KUKA KRL program: EPS_2_251825_SA38_A_20260116064124.src

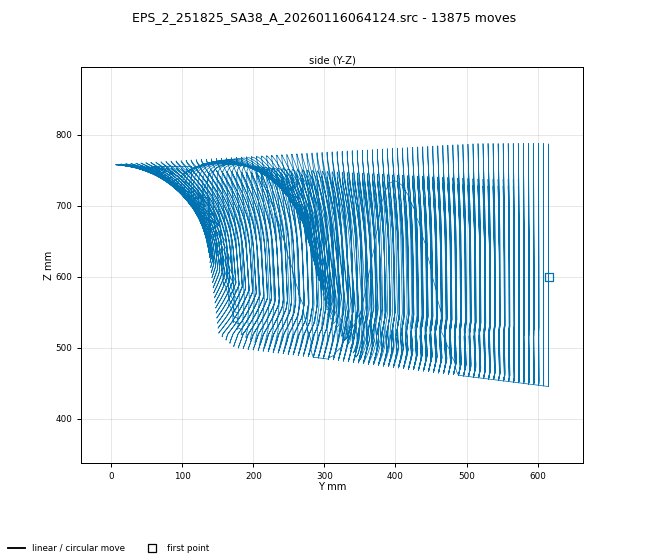
[picture p0: tool path of EPS_2_251825_SA38_A_20260116064124.src, 13875 of 13877 moves have a stored position in this frame; points joined in program order, loops and branches not executed]
&ACCESS RVP
&REL 4
&COMMENT QRS 19112012
&PARAM EDITMASK = *
DEF PART()
EXT BAS (BAS_COMMAND :IN,REAL :IN )
INT I
BAS (#INITMOV,0 )

;KUKA QRS Post kuka4.cps  Date:22-06-2017 !

File_ID=2982

QRS_PRE_INIT()

;Init var - Until changes are made in qrs_pre_init
Outlet_Square_prg=0
Inlet_1_Square_prg=0
Inlet_2_Square_prg=0
Inlet_3_Square_prg=0
Inlet_4_Square_prg=0
Inlet_5_Square_prg=0

Outlet_1={X 0.000, Y 516.340, Z 662.000, B 0.000, E1 0.000 }
Inlet_1={X 0.000, Y 523.470, Z 627.000, B 0.000, E1 180.000 }
Inlet_2={X 0.000, Y 522.780, Z 636.710, B 0.000, E1 270.000 }
Outlet_1_type=251
Inlet_1_type=201
Inlet_2_type=201
;QRS#1=Sidecore dimensions
;QRS#2=250-10" PVC SDR 35
;QRS#3=200-8" PVC SDR 35
;QRS#4=200-8" PVC SDR 35
;QRS#5=
;QRS#6=
;QRS#7=
;QRS#8=
;QRS#9=14M PSX
;QRS#10=12-08 PSX
;QRS#11=12-08 PSX
;QRS#12=
;QRS#13=
;QRS#14=
;QRS#15=
;QRS#16=1220x127x1067 3,5'
;QRS#17=EPS Height
;QRS#18=787,5
;QRS#19=*
;QRS#20= UPDATED VERSION 22-06-2017
;QRS#21=*
Outlet_Square=0100
Inlet_1_Square=0100
Inlet_2_Square=0100
Inlet_3_Square=0
Inlet_4_Square=0
Inlet_5_Square=0
Mill_Square=1
Outlet_Square_Prg=205
Inlet_1_Square_prg=204
Inlet_2_Square_prg=204

QRS_INIT()

$ADVANCE=5

; T1
PTP {E1 173.593,E2 173.593}
PTP {X 0,Y 615.508,A -85,B 0,C 180,E1 173.593,E2 173.593,E3 0,E4 0,E5 0,E6 0}
QRS_SPEED_INIT()
LIN {X 0,Y 615.508,Z 600,A -85,B 0,C 180,E1 173.593,E2 173.593,E3 0,E4 0,E5 0,E6 0} C_VEL
LIN {X 0,Y 615.508,Z 455.497,A -85,B 0,C 180,E1 173.593,E2 173.593} C_VEL
LIN {X 0,Y 615.508,Z 447.326,A -85,B 0,C 180,E1 173.593,E2 173.593} C_VEL
LIN {X 0,Y 615.49,Z 445.326,A -85,B 0,C 180,E1 173.407,E2 173.407} C_VEL
LIN {X 0,Y 615.479,Z 445.312,A -85,B 0,C 180,E1 170.801,E2 170.801} C_VEL
LIN {X 0,Y 615.481,Z 445.31,A -85,B 0,C 180,E1 168.139,E2 168.139} C_VEL
LIN {X 0,Y 615.49,Z 445.327,A -85,B 0,C 180,E1 165.451,E2 165.451} C_VEL
LIN {X 0,Y 615.478,Z 445.31,A -85,B 0,C 180,E1 162.729,E2 162.729} C_VEL
LIN {X 0,Y 615.48,Z 445.314,A -85,B 0,C 180,E1 159.967,E2 159.967} C_VEL
LIN {X 0,Y 615.483,Z 445.318,A -85,B 0,C 180,E1 157.155,E2 157.155} C_VEL
LIN {X 0,Y 615.494,Z 445.306,A -85,B 0,C 180,E1 154.284,E2 154.284} C_VEL
LIN {X 0,Y 615.489,Z 445.322,A -85,B 0,C 180,E1 151.342,E2 151.342} C_VEL
LIN {X 0,Y 615.477,Z 445.313,A -85,B 0,C 180,E1 148.913,E2 148.913} C_VEL
LIN {X 0,Y 615.485,Z 445.307,A -85,B 0,C 180,E1 146.464,E2 146.464} C_VEL
LIN {X 0,Y 615.487,Z 445.325,A -85,B 0,C 180,E1 143.575,E2 143.575} C_VEL
LIN {X 0,Y 615.479,Z 445.313,A -85,B 0,C 180,E1 140.937,E2 140.937} C_VEL
LIN {X 0,Y 615.482,Z 445.308,A -85,B 0,C 180,E1 138.525,E2 138.525} C_VEL
LIN {X 0,Y 615.485,Z 445.317,A -85,B 0,C 180,E1 135.85,E2 135.85} C_VEL
LIN {X 0,Y 615.485,Z 445.313,A -85,B 0,C 180,E1 133.047,E2 133.047} C_VEL
LIN {X 0,Y 615.478,Z 445.309,A -85,B 0,C 180,E1 130.606,E2 130.606} C_VEL
LIN {X 0,Y 615.491,Z 445.312,A -85,B 0,C 180,E1 128.012,E2 128.012} C_VEL
LIN {X 0,Y 615.496,Z 445.324,A -85,B 0,C 180,E1 125.614,E2 125.614} C_VEL
LIN {X 0,Y 615.491,Z 445.316,A -85,B 0,C 180,E1 123.235,E2 123.235} C_VEL
LIN {X 0,Y 615.479,Z 445.312,A -85,B 0,C 180,E1 120.919,E2 120.919} C_VEL
LIN {X 0,Y 615.481,Z 445.309,A -85,B 0,C 180,E1 118.449,E2 118.449} C_VEL
LIN {X 0,Y 615.499,Z 445.325,A -85,B 0,C 180,E1 115.57,E2 115.57} C_VEL
LIN {X 0,Y 615.48,Z 445.31,A -85,B 0,C 180,E1 112.844,E2 112.844} C_VEL
LIN {X 0,Y 615.485,Z 445.416,A -85,B 0,C 180,E1 112.265,E2 112.265} C_VEL
LIN {X 0,Y 615.476,Z 465.419,A -85,B 0,C 180,E1 109.511,E2 109.511} C_VEL
LIN {X 0,Y 615.479,Z 485.735,A -85,B 0,C 180,E1 106.757,E2 106.757} C_VEL
LIN {X 0,Y 615.493,Z 506.841,A -85,B 0,C 180,E1 103.933,E2 103.933} C_VEL
LIN {X 0,Y 615.482,Z 515.432,A -85,B 0,C 180,E1 102.823,E2 102.823} C_VEL
LIN {X 0,Y 615.477,Z 623.203,A -85,B 0,C 180,E1 101.547,E2 101.547} C_VEL
LIN {X 0,Y 615.485,Z 635.76,A -85,B 0,C 180,E1 101.276,E2 101.276} C_VEL
LIN {X 0,Y 615.488,Z 649.105,A -85,B 0,C 180,E1 100.842,E2 100.842} C_VEL
LIN {X 0,Y 615.491,Z 660.086,A -85,B 0,C 180,E1 100.36,E2 100.36} C_VEL
LIN {X 0,Y 615.489,Z 671.819,A -85,B 0,C 180,E1 99.695,E2 99.695} C_VEL
LIN {X 0,Y 615.499,Z 682.28,A -85,B 0,C 180,E1 98.949,E2 98.949} C_VEL
LIN {X 0,Y 615.498,Z 690.84,A -85,B 0,C 180,E1 98.205,E2 98.205} C_VEL
LIN {X 0,Y 615.497,Z 698.718,A -85,B 0,C 180,E1 97.38,E2 97.38} C_VEL
LIN {X 0,Y 615.497,Z 706.405,A -85,B 0,C 180,E1 96.391,E2 96.391} C_VEL
LIN {X 0,Y 615.497,Z 713.463,A -85,B 0,C 180,E1 95.24,E2 95.24} C_VEL
LIN {X 0,Y 615.494,Z 718.162,A -85,B 0,C 180,E1 94.256,E2 94.256} C_VEL
LIN {X 0,Y 615.494,Z 721.757,A -85,B 0,C 180,E1 93.272,E2 93.272} C_VEL
LIN {X 0,Y 615.496,Z 723.617,A -85,B 0,C 180,E1 92.617,E2 92.617} C_VEL
LIN {X 0,Y 615.498,Z 725.035,A -85,B 0,C 180,E1 91.962,E2 91.962} C_VEL
LIN {X 0,Y 615.496,Z 726.642,A -85,B 0,C 180,E1 90.653,E2 90.653} C_VEL
LIN {X 0,Y 615.495,Z 726.884,A -85,B 0,C 180,E1 89.999,E2 89.999} C_VEL
LIN {X 0,Y 615.495,Z 726.705,A -85,B 0,C 180,E1 89.345,E2 89.345} C_VEL
LIN {X 0,Y 615.499,Z 725.181,A -85,B 0,C 180,E1 88.036,E2 88.036} C_VEL
LIN {X 0,Y 615.498,Z 723.839,A -85,B 0,C 180,E1 87.381,E2 87.381} C_VEL
LIN {X 0,Y 615.496,Z 720.991,A -85,B 0,C 180,E1 86.399,E2 86.399} C_VEL
LIN {X 0,Y 615.498,Z 717.131,A -85,B 0,C 180,E1 85.415,E2 85.415} C_VEL
LIN {X 0,Y 615.498,Z 712.147,A -85,B 0,C 180,E1 84.43,E2 84.43} C_VEL
LIN {X 0,Y 615.496,Z 705.708,A -85,B 0,C 180,E1 83.418,E2 83.418} C_VEL
LIN {X 0,Y 615.497,Z 698.03,A -85,B 0,C 180,E1 82.454,E2 82.454} C_VEL
LIN {X 0,Y 615.498,Z 688.25,A -85,B 0,C 180,E1 81.463,E2 81.463} C_VEL
LIN {X 0,Y 615.498,Z 677.982,A -85,B 0,C 180,E1 80.635,E2 80.635} C_VEL
LIN {X 0,Y 615.493,Z 666.416,A -85,B 0,C 180,E1 79.888,E2 79.888} C_VEL
LIN {X 0,Y 615.496,Z 654.517,A -85,B 0,C 180,E1 79.291,E2 79.291} C_VEL
LIN {X 0,Y 615.489,Z 641.636,A -85,B 0,C 180,E1 78.806,E2 78.806} C_VEL
LIN {X 0,Y 615.477,Z 629.028,A -85,B 0,C 180,E1 78.472,E2 78.472} C_VEL
LIN {X 0,Y 615.479,Z 615.873,A -85,B 0,C 180,E1 78.264,E2 78.264} C_VEL
LIN {X 0,Y 615.488,Z 515.092,A -85,B 0,C 180,E1 77.071,E2 77.071} C_VEL
LIN {X 0,Y 615.479,Z 494.007,A -85,B 0,C 180,E1 74.264,E2 74.264} C_VEL
LIN {X 0,Y 615.484,Z 473.933,A -85,B 0,C 180,E1 71.559,E2 71.559} C_VEL
LIN {X 0,Y 615.493,Z 453.348,A -85,B 0,C 180,E1 68.743,E2 68.743} C_VEL
LIN {X 0,Y 615.479,Z 445.31,A -85,B 0,C 180,E1 67.625,E2 67.625} C_VEL
LIN {X 0,Y 615.488,Z 445.309,A -85,B 0,C 180,E1 65.008,E2 65.008} C_VEL
LIN {X 0,Y 615.495,Z 445.317,A -85,B 0,C 180,E1 62.085,E2 62.085} C_VEL
LIN {X 0,Y 615.499,Z 445.31,A -85,B 0,C 180,E1 59.84,E2 59.84} C_VEL
LIN {X 0,Y 615.481,Z 445.309,A -85,B 0,C 180,E1 57.541,E2 57.541} C_VEL
LIN {X 0,Y 615.478,Z 445.309,A -85,B 0,C 180,E1 55.184,E2 55.184} C_VEL
LIN {X 0,Y 615.493,Z 445.312,A -85,B 0,C 180,E1 52.758,E2 52.758} C_VEL
LIN {X 0,Y 615.495,Z 445.313,A -85,B 0,C 180,E1 49.911,E2 49.911} C_VEL
LIN {X 0,Y 615.49,Z 445.308,A -85,B 0,C 180,E1 47.647,E2 47.647} C_VEL
LIN {X 0,Y 615.481,Z 445.311,A -85,B 0,C 180,E1 44.93,E2 44.93} C_VEL
LIN {X 0,Y 615.49,Z 445.319,A -85,B 0,C 180,E1 42.08,E2 42.08} C_VEL
LIN {X 0,Y 615.499,Z 445.308,A -85,B 0,C 180,E1 39.75,E2 39.75} C_VEL
LIN {X 0,Y 615.479,Z 445.312,A -85,B 0,C 180,E1 36.935,E2 36.935} C_VEL
LIN {X 0,Y 615.493,Z 445.313,A -85,B 0,C 180,E1 34.701,E2 34.701} C_VEL
LIN {X 0,Y 615.488,Z 445.31,A -85,B 0,C 180,E1 31.686,E2 31.686} C_VEL
LIN {X 0,Y 615.482,Z 445.308,A -85,B 0,C 180,E1 29.407,E2 29.407} C_VEL
LIN {X 0,Y 615.478,Z 445.31,A -85,B 0,C 180,E1 27.042,E2 27.042} C_VEL
LIN {X 0,Y 615.494,Z 445.325,A -85,B 0,C 180,E1 24.272,E2 24.272} C_VEL
LIN {X 0,Y 615.476,Z 445.317,A -85,B 0,C 180,E1 23.023,E2 23.023} C_VEL
LIN {X 0,Y 615.48,Z 466.086,A -85,B 0,C 180,E1 20.295,E2 20.295} C_VEL
LIN {X 0,Y 615.487,Z 488.175,A -85,B 0,C 180,E1 17.442,E2 17.442} C_VEL
LIN {X 0,Y 615.488,Z 510.904,A -85,B 0,C 180,E1 14.549,E2 14.549} C_VEL
LIN {X 0,Y 615.481,Z 524.429,A -85,B 0,C 180,E1 12.845,E2 12.845} C_VEL
LIN {X 0,Y 615.489,Z 633.994,A -85,B 0,C 180,E1 11.527,E2 11.527} C_VEL
LIN {X 0,Y 615.483,Z 646.945,A -85,B 0,C 180,E1 11.235,E2 11.235} C_VEL
LIN {X 0,Y 615.49,Z 658.842,A -85,B 0,C 180,E1 10.841,E2 10.841} C_VEL
LIN {X 0,Y 615.481,Z 671.405,A -85,B 0,C 180,E1 10.278,E2 10.278} C_VEL
LIN {X 0,Y 615.493,Z 682.784,A -85,B 0,C 180,E1 9.613,E2 9.613} C_VEL
LIN {X 0,Y 615.498,Z 693.031,A -85,B 0,C 180,E1 8.868,E2 8.868} C_VEL
LIN {X 0,Y 615.498,Z 702.243,A -85,B 0,C 180,E1 8.041,E2 8.041} C_VEL
LIN {X 0,Y 615.499,Z 711.101,A -85,B 0,C 180,E1 7.057,E2 7.057} C_VEL
LIN {X 0,Y 615.497,Z 718.333,A -85,B 0,C 180,E1 6.063,E2 6.063} C_VEL
LIN {X 0,Y 615.497,Z 723.167,A -85,B 0,C 180,E1 5.241,E2 5.241} C_VEL
LIN {X 0,Y 615.493,Z 727.867,A -85,B 0,C 180,E1 4.257,E2 4.257} C_VEL
LIN {X 0,Y 615.495,Z 731.464,A -85,B 0,C 180,E1 3.273,E2 3.273} C_VEL
LIN {X 0,Y 615.496,Z 733.324,A -85,B 0,C 180,E1 2.618,E2 2.618} C_VEL
LIN {X 0,Y 615.497,Z 734.743,A -85,B 0,C 180,E1 1.963,E2 1.963} C_VEL
LIN {X 0,Y 615.496,Z 736.351,A -85,B 0,C 180,E1 0.654,E2 0.654} C_VEL
LIN {X 0,Y 615.494,Z 736.594,A -85,B 0,C 180,E1 0,E2 0} C_VEL
LIN {X 0,Y 615.496,Z 736.415,A -85,B 0,C 180,E1 -0.654,E2 -0.654} C_VEL
LIN {X 0,Y 615.496,Z 734.893,A -85,B 0,C 180,E1 -1.963,E2 -1.963} C_VEL
LIN {X 0,Y 615.498,Z 733.551,A -85,B 0,C 180,E1 -2.618,E2 -2.618} C_VEL
LIN {X 0,Y 615.496,Z 730.704,A -85,B 0,C 180,E1 -3.601,E2 -3.601} C_VEL
LIN {X 0,Y 615.499,Z 726.844,A -85,B 0,C 180,E1 -4.584,E2 -4.584} C_VEL
LIN {X 0,Y 615.498,Z 721.862,A -85,B 0,C 180,E1 -5.57,E2 -5.57} C_VEL
LIN {X 0,Y 615.497,Z 715.413,A -85,B 0,C 180,E1 -6.583,E2 -6.583} C_VEL
LIN {X 0,Y 615.497,Z 707.747,A -85,B 0,C 180,E1 -7.545,E2 -7.545} C_VEL
LIN {X 0,Y 615.498,Z 697.969,A -85,B 0,C 180,E1 -8.536,E2 -8.536} C_VEL
LIN {X 0,Y 615.497,Z 687.704,A -85,B 0,C 180,E1 -9.364,E2 -9.364} C_VEL
LIN {X 0,Y 615.476,Z 676.143,A -85,B 0,C 180,E1 -10.111,E2 -10.111} C_VEL
LIN {X 0,Y 615.497,Z 664.291,A -85,B 0,C 180,E1 -10.707,E2 -10.707} C_VEL
LIN {X 0,Y 615.478,Z 651.373,A -85,B 0,C 180,E1 -11.193,E2 -11.193} C_VEL
LIN {X 0,Y 615.486,Z 638.772,A -85,B 0,C 180,E1 -11.527,E2 -11.527} C_VEL
LIN {X 0,Y 615.487,Z 625.651,A -85,B 0,C 180,E1 -11.735,E2 -11.735} C_VEL
LIN {X 0,Y 615.478,Z 524.479,A -85,B 0,C 180,E1 -12.929,E2 -12.929} C_VEL
LIN {X 0,Y 615.488,Z 502.257,A -85,B 0,C 180,E1 -15.735,E2 -15.735} C_VEL
LIN {X 0,Y 615.492,Z 479.506,A -85,B 0,C 180,E1 -18.646,E2 -18.646} C_VEL
LIN {X 0,Y 615.485,Z 456.727,A -85,B 0,C 180,E1 -21.608,E2 -21.608} C_VEL
LIN {X 0,Y 615.476,Z 445.312,A -85,B 0,C 180,E1 -23.134,E2 -23.134} C_VEL
LIN {X 0,Y 615.496,Z 445.309,A -85,B 0,C 180,E1 -25.715,E2 -25.715} C_VEL
LIN {X 0,Y 615.49,Z 445.314,A -85,B 0,C 180,E1 -28.658,E2 -28.658} C_VEL
LIN {X 0,Y 615.477,Z 445.31,A -85,B 0,C 180,E1 -31.084,E2 -31.084} C_VEL
LIN {X 0,Y 615.486,Z 445.312,A -85,B 0,C 180,E1 -33.533,E2 -33.533} C_VEL
LIN {X 0,Y 615.49,Z 445.315,A -85,B 0,C 180,E1 -36.425,E2 -36.425} C_VEL
LIN {X 0,Y 615.479,Z 445.31,A -85,B 0,C 180,E1 -39.06,E2 -39.06} C_VEL
LIN {X 0,Y 615.482,Z 445.315,A -85,B 0,C 180,E1 -41.474,E2 -41.474} C_VEL
LIN {X 0,Y 615.479,Z 445.319,A -85,B 0,C 180,E1 -44.15,E2 -44.15} C_VEL
LIN {X 0,Y 615.486,Z 445.309,A -85,B 0,C 180,E1 -46.953,E2 -46.953} C_VEL
LIN {X 0,Y 615.489,Z 445.32,A -85,B 0,C 180,E1 -49.911,E2 -49.911} C_VEL
LIN {X 0,Y 615.49,Z 445.308,A -85,B 0,C 180,E1 -52.757,E2 -52.757} C_VEL
LIN {X 0,Y 615.488,Z 445.319,A -85,B 0,C 180,E1 -55.299,E2 -55.299} C_VEL
LIN {X 0,Y 615.496,Z 445.32,A -85,B 0,C 180,E1 -57.668,E2 -57.668} C_VEL
LIN {X 0,Y 615.478,Z 445.311,A -85,B 0,C 180,E1 -60.593,E2 -60.593} C_VEL
LIN {X 0,Y 615.496,Z 445.313,A -85,B 0,C 180,E1 -62.954,E2 -62.954} C_VEL
LIN {X 0,Y 615.493,Z 445.313,A -85,B 0,C 180,E1 -65.728,E2 -65.728} C_VEL
LIN {X 0,Y 615.475,Z 445.416,A -85,B 0,C 180,E1 -66.4,E2 -66.4} C_VEL
LIN {X 0,Y 615.49,Z 471.23,A -85,B 0,C 180,E1 -69.094,E2 -69.094} C_VEL
LIN {X 0,Y 615.484,Z 498.445,A -85,B 0,C 180,E1 -71.882,E2 -71.882} C_VEL
LIN {X 0,Y 615.492,Z 523.292,A -85,B 0,C 180,E1 -74.392,E2 -74.392} C_VEL
LIN {X 0,Y 615.484,Z 662.17,A -85,B 0,C 180,E1 -76.05,E2 -76.05} C_VEL
LIN {X 0,Y 615.486,Z 675.829,A -85,B 0,C 180,E1 -76.336,E2 -76.336} C_VEL
LIN {X 0,Y 615.496,Z 689.547,A -85,B 0,C 180,E1 -76.756,E2 -76.756} C_VEL
LIN {X 0,Y 615.497,Z 702.821,A -85,B 0,C 180,E1 -77.302,E2 -77.302} C_VEL
LIN {X 0,Y 615.492,Z 715.587,A -85,B 0,C 180,E1 -77.971,E2 -77.971} C_VEL
LIN {X 0,Y 615.499,Z 727.172,A -85,B 0,C 180,E1 -78.723,E2 -78.723} C_VEL
LIN {X 0,Y 615.498,Z 738.739,A -85,B 0,C 180,E1 -79.639,E2 -79.639} C_VEL
LIN {X 0,Y 615.497,Z 749.081,A -85,B 0,C 180,E1 -80.635,E2 -80.635} C_VEL
LIN {X 0,Y 615.497,Z 757.596,A -85,B 0,C 180,E1 -81.628,E2 -81.628} C_VEL
LIN {X 0,Y 615.496,Z 765.722,A -85,B 0,C 180,E1 -82.784,E2 -82.784} C_VEL
LIN {X 0,Y 615.496,Z 771.426,A -85,B 0,C 180,E1 -83.772,E2 -83.772} C_VEL
LIN {X 0,Y 615.495,Z 776.077,A -85,B 0,C 180,E1 -84.758,E2 -84.758} C_VEL
LIN {X 0,Y 615.494,Z 780.899,A -85,B 0,C 180,E1 -86.071,E2 -86.071} C_VEL
LIN {X 0,Y 615.496,Z 784.25,A -85,B 0,C 180,E1 -87.381,E2 -87.381} C_VEL
LIN {X 0,Y 615.489,Z 786.228,A -85,B 0,C 180,E1 -88.691,E2 -88.691} C_VEL
LIN {X 0,Y 615.493,Z 786.889,A -85,B 0,C 180,E1 -89.999,E2 -89.999} C_VEL
LIN {X 0,Y 615.489,Z 786.23,A -85,B 0,C 180,E1 -91.308,E2 -91.308} C_VEL
LIN {X 0,Y 615.496,Z 784.254,A -85,B 0,C 180,E1 -92.617,E2 -92.617} C_VEL
LIN {X 0,Y 615.493,Z 780.904,A -85,B 0,C 180,E1 -93.928,E2 -93.928} C_VEL
LIN {X 0,Y 615.495,Z 776.084,A -85,B 0,C 180,E1 -95.24,E2 -95.24} C_VEL
LIN {X 0,Y 615.495,Z 769.633,A -85,B 0,C 180,E1 -96.556,E2 -96.556} C_VEL
LIN {X 0,Y 615.497,Z 762.447,A -85,B 0,C 180,E1 -97.709,E2 -97.709} C_VEL
LIN {X 0,Y 615.497,Z 754.911,A -85,B 0,C 180,E1 -98.701,E2 -98.701} C_VEL
LIN {X 0,Y 615.495,Z 745.862,A -85,B 0,C 180,E1 -99.695,E2 -99.695} C_VEL
LIN {X 0,Y 615.497,Z 735.765,A -85,B 0,C 180,E1 -100.617,E2 -100.617} C_VEL
LIN {X 0,Y 615.498,Z 724.871,A -85,B 0,C 180,E1 -101.442,E2 -101.442} C_VEL
LIN {X 0,Y 615.488,Z 712.724,A -85,B 0,C 180,E1 -102.194,E2 -102.194} C_VEL
LIN {X 0,Y 615.495,Z 699.113,A -85,B 0,C 180,E1 -102.864,E2 -102.864} C_VEL
LIN {X 0,Y 615.492,Z 685.864,A -85,B 0,C 180,E1 -103.368,E2 -103.368} C_VEL
LIN {X 0,Y 615.484,Z 672.328,A -85,B 0,C 180,E1 -103.747,E2 -103.747} C_VEL
LIN {X 0,Y 615.486,Z 658.097,A -85,B 0,C 180,E1 -104.008,E2 -104.008} C_VEL
LIN {X 0,Y 615.493,Z 523.098,A -85,B 0,C 180,E1 -105.628,E2 -105.628} C_VEL
LIN {X 0,Y 615.479,Z 495.289,A -85,B 0,C 180,E1 -108.44,E2 -108.44} C_VEL
LIN {X 0,Y 615.496,Z 467.859,A -85,B 0,C 180,E1 -111.255,E2 -111.255} C_VEL
LIN {X 0,Y 615.477,Z 445.31,A -85,B 0,C 180,E1 -113.612,E2 -113.612} C_VEL
LIN {X 0,Y 615.492,Z 445.317,A -85,B 0,C 180,E1 -116.443,E2 -116.443} C_VEL
LIN {X 0,Y 615.493,Z 445.324,A -85,B 0,C 180,E1 -118.656,E2 -118.656} C_VEL
LIN {X 0,Y 615.493,Z 445.314,A -85,B 0,C 180,E1 -121.087,E2 -121.087} C_VEL
LIN {X 0,Y 615.479,Z 445.31,A -85,B 0,C 180,E1 -123.533,E2 -123.533} C_VEL
LIN {X 0,Y 615.477,Z 445.31,A -85,B 0,C 180,E1 -125.832,E2 -125.832} C_VEL
LIN {X 0,Y 615.488,Z 445.31,A -85,B 0,C 180,E1 -128.067,E2 -128.067} C_VEL
LIN {X 0,Y 615.49,Z 445.314,A -85,B 0,C 180,E1 -131.095,E2 -131.095} C_VEL
LIN {X 0,Y 615.499,Z 445.308,A -85,B 0,C 180,E1 -133.242,E2 -133.242} C_VEL
LIN {X 0,Y 615.482,Z 445.31,A -85,B 0,C 180,E1 -136.001,E2 -136.001} C_VEL
LIN {X 0,Y 615.492,Z 445.318,A -85,B 0,C 180,E1 -138.903,E2 -138.903} C_VEL
LIN {X 0,Y 615.487,Z 445.314,A -85,B 0,C 180,E1 -141.096,E2 -141.096} C_VEL
LIN {X 0,Y 615.481,Z 445.308,A -85,B 0,C 180,E1 -143.575,E2 -143.575} C_VEL
LIN {X 0,Y 615.496,Z 445.319,A -85,B 0,C 180,E1 -146.462,E2 -146.462} C_VEL
LIN {X 0,Y 615.49,Z 445.313,A -85,B 0,C 180,E1 -149.08,E2 -149.08} C_VEL
LIN {X 0,Y 615.483,Z 445.308,A -85,B 0,C 180,E1 -151.548,E2 -151.548} C_VEL
LIN {X 0,Y 615.493,Z 445.319,A -85,B 0,C 180,E1 -154.427,E2 -154.427} C_VEL
LIN {X 0,Y 615.486,Z 445.312,A -85,B 0,C 180,E1 -157.155,E2 -157.155} C_VEL
LIN {X 0,Y 615.487,Z 445.308,A -85,B 0,C 180,E1 -159.439,E2 -159.439} C_VEL
LIN {X 0,Y 615.478,Z 445.313,A -85,B 0,C 180,E1 -162.043,E2 -162.043} C_VEL
LIN {X 0,Y 615.489,Z 445.321,A -85,B 0,C 180,E1 -164.774,E2 -164.774} C_VEL
LIN {X 0,Y 615.49,Z 445.307,A -85,B 0,C 180,E1 -167.47,E2 -167.47} C_VEL
LIN {X 0,Y 615.479,Z 445.315,A -85,B 0,C 180,E1 -170.138,E2 -170.138} C_VEL
LIN {X 0,Y 615.486,Z 445.321,A -85,B 0,C 180,E1 -172.784,E2 -172.784} C_VEL
LIN {X 0,Y 615.496,Z 445.306,A -85,B 0,C 180,E1 -175.416,E2 -175.416} C_VEL
LIN {X 0,Y 615.477,Z 445.314,A -85,B 0,C 180,E1 -178.037,E2 -178.037} C_VEL
LIN {X 0,Y 615.488,Z 445.325,A -85,B 0,C 180,E1 -180.654,E2 -180.654} C_VEL
LIN {X 0,Y 615.484,Z 445.31,A -85,B 0,C 180,E1 -183.273,E2 -183.273} C_VEL
LIN {X 0,Y 615.478,Z 445.311,A -85,B 0,C 180,E1 -185.899,E2 -185.899} C_VEL
LIN {X 0,Y 615.49,Z 445.326,A -85,B 0,C 180,E1 -186.593,E2 -186.593} C_VEL
LIN {X 0,Y 614.808,Z 445.46,A -85,B 0,C 180,E1 -187.138,E2 -187.138} C_VEL
LIN {X 0,Y 611.967,Z 445.877,A -85,B 0,C 180,E1 -188.024,E2 -188.024} C_VEL
LIN {X 0,Y 609.574,Z 446.186,A -85,B 0,C 180,E1 -188.737,E2 -188.737} C_VEL
LIN {X 0,Y 608.54,Z 446.303,A -85,B 0,C 180,E1 -189.287,E2 -189.287} C_VEL
LIN {X 0,Y 608.451,Z 446.312,A -85,B 0,C 180,E1 -189.473,E2 -189.473} C_VEL
LIN {X 0,Y 608.458,Z 446.314,A -85,B 0,C 180,E1 -192,E2 -192} C_VEL
LIN {X 0,Y 608.474,Z 446.317,A -85,B 0,C 180,E1 -194.721,E2 -194.721} C_VEL
LIN {X 0,Y 608.445,Z 446.313,A -85,B 0,C 180,E1 -197.477,E2 -197.477} C_VEL
LIN {X 0,Y 608.461,Z 446.317,A -85,B 0,C 180,E1 -200.274,E2 -200.274} C_VEL
LIN {X 0,Y 608.447,Z 446.315,A -85,B 0,C 180,E1 -203.124,E2 -203.124} C_VEL
LIN {X 0,Y 608.476,Z 446.31,A -85,B 0,C 180,E1 -205.725,E2 -205.725} C_VEL
LIN {X 0,Y 608.476,Z 446.318,A -85,B 0,C 180,E1 -208.623,E2 -208.623} C_VEL
LIN {X 0,Y 608.469,Z 446.31,A -85,B 0,C 180,E1 -211.317,E2 -211.317} C_VEL
LIN {X 0,Y 608.471,Z 446.31,A -85,B 0,C 180,E1 -213.737,E2 -213.737} C_VEL
LIN {X 0,Y 608.472,Z 446.314,A -85,B 0,C 180,E1 -216.091,E2 -216.091} C_VEL
LIN {X 0,Y 608.467,Z 446.32,A -85,B 0,C 180,E1 -218.588,E2 -218.588} C_VEL
LIN {X 0,Y 608.456,Z 446.312,A -85,B 0,C 180,E1 -221.344,E2 -221.344} C_VEL
LIN {X 0,Y 608.453,Z 446.319,A -85,B 0,C 180,E1 -224.265,E2 -224.265} C_VEL
LIN {X 0,Y 608.453,Z 446.314,A -85,B 0,C 180,E1 -227.042,E2 -227.042} C_VEL
LIN {X 0,Y 608.453,Z 446.313,A -85,B 0,C 180,E1 -229.698,E2 -229.698} C_VEL
LIN {X 0,Y 608.475,Z 446.317,A -85,B 0,C 180,E1 -232.256,E2 -232.256} C_VEL
LIN {X 0,Y 608.471,Z 446.311,A -85,B 0,C 180,E1 -235.092,E2 -235.092} C_VEL
LIN {X 0,Y 608.47,Z 446.312,A -85,B 0,C 180,E1 -237.907,E2 -237.907} C_VEL
LIN {X 0,Y 608.472,Z 446.317,A -85,B 0,C 180,E1 -240.222,E2 -240.222} C_VEL
LIN {X 0,Y 608.483,Z 446.313,A -85,B 0,C 180,E1 -242.793,E2 -242.793} C_VEL
LIN {X 0,Y 608.455,Z 446.312,A -85,B 0,C 180,E1 -245.43,E2 -245.43} C_VEL
LIN {X 0,Y 608.476,Z 446.356,A -85,B 0,C 180,E1 -247.596,E2 -247.596} C_VEL
LIN {X 0,Y 608.536,Z 462.894,A -85,B 0,C 180,E1 -249.906,E2 -249.906} C_VEL
LIN {X 0,Y 608.527,Z 483.248,A -85,B 0,C 180,E1 -252.7,E2 -252.7} C_VEL
LIN {X 0,Y 608.509,Z 506.148,A -85,B 0,C 180,E1 -255.794,E2 -255.794} C_VEL
LIN {X 0,Y 608.481,Z 515.512,A -85,B 0,C 180,E1 -257.027,E2 -257.027} C_VEL
LIN {X 0,Y 608.541,Z 623.349,A -85,B 0,C 180,E1 -258.32,E2 -258.32} C_VEL
LIN {X 0,Y 608.525,Z 636.65,A -85,B 0,C 180,E1 -258.615,E2 -258.615} C_VEL
LIN {X 0,Y 608.52,Z 649.964,A -85,B 0,C 180,E1 -259.059,E2 -259.059} C_VEL
LIN {X 0,Y 608.501,Z 661.886,A -85,B 0,C 180,E1 -259.604,E2 -259.604} C_VEL
LIN {X 0,Y 608.502,Z 673.304,A -85,B 0,C 180,E1 -260.276,E2 -260.276} C_VEL
LIN {X 0,Y 608.474,Z 683.596,A -85,B 0,C 180,E1 -261.03,E2 -261.03} C_VEL
LIN {X 0,Y 608.464,Z 692.859,A -85,B 0,C 180,E1 -261.867,E2 -261.867} C_VEL
LIN {X 0,Y 608.466,Z 701.831,A -85,B 0,C 180,E1 -262.868,E2 -262.868} C_VEL
LIN {X 0,Y 608.444,Z 709.061,A -85,B 0,C 180,E1 -263.867,E2 -263.867} C_VEL
LIN {X 0,Y 608.462,Z 713.939,A -85,B 0,C 180,E1 -264.699,E2 -264.699} C_VEL
LIN {X 0,Y 608.439,Z 718.682,A -85,B 0,C 180,E1 -265.695,E2 -265.695} C_VEL
LIN {X 0,Y 608.425,Z 722.315,A -85,B 0,C 180,E1 -266.69,E2 -266.69} C_VEL
LIN {X 0,Y 608.425,Z 724.193,A -85,B 0,C 180,E1 -267.353,E2 -267.353} C_VEL
LIN {X 0,Y 608.443,Z 725.628,A -85,B 0,C 180,E1 -268.015,E2 -268.015} C_VEL
LIN {X 0,Y 608.439,Z 727.252,A -85,B 0,C 180,E1 -269.339,E2 -269.339} C_VEL
LIN {X 0,Y 608.435,Z 727.496,A -85,B 0,C 180,E1 -270.001,E2 -270.001} C_VEL
LIN {X 0,Y 608.438,Z 727.314,A -85,B 0,C 180,E1 -270.663,E2 -270.663} C_VEL
LIN {X 0,Y 608.444,Z 725.775,A -85,B 0,C 180,E1 -271.987,E2 -271.987} C_VEL
LIN {X 0,Y 608.426,Z 724.417,A -85,B 0,C 180,E1 -272.649,E2 -272.649} C_VEL
LIN {X 0,Y 608.45,Z 721.539,A -85,B 0,C 180,E1 -273.643,E2 -273.643} C_VEL
LIN {X 0,Y 608.433,Z 717.639,A -85,B 0,C 180,E1 -274.639,E2 -274.639} C_VEL
LIN {X 0,Y 608.449,Z 712.608,A -85,B 0,C 180,E1 -275.635,E2 -275.635} C_VEL
LIN {X 0,Y 608.441,Z 706.289,A -85,B 0,C 180,E1 -276.634,E2 -276.634} C_VEL
LIN {X 0,Y 608.476,Z 698.371,A -85,B 0,C 180,E1 -277.634,E2 -277.634} C_VEL
LIN {X 0,Y 608.472,Z 688.528,A -85,B 0,C 180,E1 -278.637,E2 -278.637} C_VEL
LIN {X 0,Y 608.48,Z 678.203,A -85,B 0,C 180,E1 -279.474,E2 -279.474} C_VEL
LIN {X 0,Y 608.49,Z 666.586,A -85,B 0,C 180,E1 -280.23,E2 -280.23} C_VEL
LIN {X 0,Y 608.528,Z 655.367,A -85,B 0,C 180,E1 -280.803,E2 -280.803} C_VEL
LIN {X 0,Y 608.527,Z 642.838,A -85,B 0,C 180,E1 -281.288,E2 -281.288} C_VEL
LIN {X 0,Y 608.522,Z 630.026,A -85,B 0,C 180,E1 -281.64,E2 -281.64} C_VEL
LIN {X 0,Y 608.533,Z 617.733,A -85,B 0,C 180,E1 -281.851,E2 -281.851} C_VEL
LIN {X 0,Y 608.529,Z 515.793,A -85,B 0,C 180,E1 -283.058,E2 -283.058} C_VEL
LIN {X 0,Y 608.466,Z 515.079,A -85,B 0,C 180,E1 -283.102,E2 -283.102} C_VEL
LIN {X 0,Y 608.488,Z 495.351,A -85,B 0,C 180,E1 -285.75,E2 -285.75} C_VEL
LIN {X 0,Y 608.529,Z 475.149,A -85,B 0,C 180,E1 -288.496,E2 -288.496} C_VEL
LIN {X 0,Y 608.568,Z 454.621,A -85,B 0,C 180,E1 -291.333,E2 -291.333} C_VEL
LIN {X 0,Y 608.465,Z 446.313,A -85,B 0,C 180,E1 -292.527,E2 -292.527} C_VEL
LIN {X 0,Y 608.456,Z 446.312,A -85,B 0,C 180,E1 -294.572,E2 -294.572} C_VEL
LIN {X 0,Y 608.485,Z 446.312,A -85,B 0,C 180,E1 -297.208,E2 -297.208} C_VEL
LIN {X 0,Y 608.477,Z 446.315,A -85,B 0,C 180,E1 -299.973,E2 -299.973} C_VEL
LIN {X 0,Y 608.458,Z 446.312,A -85,B 0,C 180,E1 -302.88,E2 -302.88} C_VEL
LIN {X 0,Y 608.447,Z 446.317,A -85,B 0,C 180,E1 -305.278,E2 -305.278} C_VEL
LIN {X 0,Y 608.477,Z 446.319,A -85,B 0,C 180,E1 -307.746,E2 -307.746} C_VEL
LIN {X 0,Y 608.453,Z 446.313,A -85,B 0,C 180,E1 -310.329,E2 -310.329} C_VEL
LIN {X 0,Y 608.453,Z 446.313,A -85,B 0,C 180,E1 -312.96,E2 -312.96} C_VEL
LIN {X 0,Y 608.462,Z 446.321,A -85,B 0,C 180,E1 -315.736,E2 -315.736} C_VEL
LIN {X 0,Y 608.457,Z 446.311,A -85,B 0,C 180,E1 -318.659,E2 -318.659} C_VEL
LIN {X 0,Y 608.472,Z 446.319,A -85,B 0,C 180,E1 -321.76,E2 -321.76} C_VEL
LIN {X 0,Y 608.449,Z 446.312,A -85,B 0,C 180,E1 -324.723,E2 -324.723} C_VEL
LIN {X 0,Y 608.469,Z 446.317,A -85,B 0,C 180,E1 -327.477,E2 -327.477} C_VEL
LIN {X 0,Y 608.477,Z 446.312,A -85,B 0,C 180,E1 -330.221,E2 -330.221} C_VEL
LIN {X 0,Y 608.473,Z 446.31,A -85,B 0,C 180,E1 -332.795,E2 -332.795} C_VEL
LIN {X 0,Y 608.455,Z 446.318,A -85,B 0,C 180,E1 -335.429,E2 -335.429} C_VEL
LIN {X 0,Y 608.475,Z 446.327,A -85,B 0,C 180,E1 -336.832,E2 -336.832} C_VEL
LIN {X 0,Y 608.584,Z 462.746,A -85,B 0,C 180,E1 -339.023,E2 -339.023} C_VEL
LIN {X 0,Y 608.533,Z 484.192,A -85,B 0,C 180,E1 -341.831,E2 -341.831} C_VEL
LIN {X 0,Y 608.497,Z 505.639,A -85,B 0,C 180,E1 -344.595,E2 -344.595} C_VEL
LIN {X 0,Y 608.488,Z 524.573,A -85,B 0,C 180,E1 -347.005,E2 -347.005} C_VEL
LIN {X 0,Y 608.554,Z 632.98,A -85,B 0,C 180,E1 -348.319,E2 -348.319} C_VEL
LIN {X 0,Y 608.531,Z 646.326,A -85,B 0,C 180,E1 -348.614,E2 -348.614} C_VEL
LIN {X 0,Y 608.511,Z 658.811,A -85,B 0,C 180,E1 -349.026,E2 -349.026} C_VEL
LIN {X 0,Y 608.509,Z 669.944,A -85,B 0,C 180,E1 -349.519,E2 -349.519} C_VEL
LIN {X 0,Y 608.488,Z 681.719,A -85,B 0,C 180,E1 -350.191,E2 -350.191} C_VEL
LIN {X 0,Y 608.485,Z 692.232,A -85,B 0,C 180,E1 -350.946,E2 -350.946} C_VEL
LIN {X 0,Y 608.475,Z 700.843,A -85,B 0,C 180,E1 -351.699,E2 -351.699} C_VEL
LIN {X 0,Y 608.471,Z 708.773,A -85,B 0,C 180,E1 -352.534,E2 -352.534} C_VEL
LIN {X 0,Y 608.468,Z 716.279,A -85,B 0,C 180,E1 -353.497,E2 -353.497} C_VEL
LIN {X 0,Y 608.451,Z 721.819,A -85,B 0,C 180,E1 -354.365,E2 -354.365} C_VEL
LIN {X 0,Y 608.431,Z 726.96,A -85,B 0,C 180,E1 -355.362,E2 -355.362} C_VEL
LIN {X 0,Y 608.45,Z 730.95,A -85,B 0,C 180,E1 -356.358,E2 -356.358} C_VEL
LIN {X 0,Y 608.425,Z 733.901,A -85,B 0,C 180,E1 -357.352,E2 -357.352} C_VEL
LIN {X 0,Y 608.442,Z 735.337,A -85,B 0,C 180,E1 -358.014,E2 -358.014} C_VEL
LIN {X 0,Y 608.439,Z 736.962,A -85,B 0,C 180,E1 -359.338,E2 -359.338} C_VEL
LIN {X 0,Y 608.434,Z 737.205,A -85,B 0,C 180,E1 -360,E2 -360} C_VEL
LIN {X 0,Y 608.439,Z 737.025,A -85,B 0,C 180,E1 -360.662,E2 -360.662} C_VEL
LIN {X 0,Y 608.441,Z 735.486,A -85,B 0,C 180,E1 -361.986,E2 -361.986} C_VEL
LIN {X 0,Y 608.426,Z 734.127,A -85,B 0,C 180,E1 -362.648,E2 -362.648} C_VEL
LIN {X 0,Y 608.449,Z 731.251,A -85,B 0,C 180,E1 -363.642,E2 -363.642} C_VEL
LIN {X 0,Y 608.433,Z 727.351,A -85,B 0,C 180,E1 -364.638,E2 -364.638} C_VEL
LIN {X 0,Y 608.449,Z 722.321,A -85,B 0,C 180,E1 -365.634,E2 -365.634} C_VEL
LIN {X 0,Y 608.442,Z 716.005,A -85,B 0,C 180,E1 -366.633,E2 -366.633} C_VEL
LIN {X 0,Y 608.475,Z 708.089,A -85,B 0,C 180,E1 -367.633,E2 -367.633} C_VEL
LIN {X 0,Y 608.472,Z 698.243,A -85,B 0,C 180,E1 -368.636,E2 -368.636} C_VEL
LIN {X 0,Y 608.48,Z 687.924,A -85,B 0,C 180,E1 -369.473,E2 -369.473} C_VEL
LIN {X 0,Y 608.473,Z 676.312,A -85,B 0,C 180,E1 -370.229,E2 -370.229} C_VEL
LIN {X 0,Y 608.525,Z 665.111,A -85,B 0,C 180,E1 -370.801,E2 -370.801} C_VEL
LIN {X 0,Y 608.527,Z 652.467,A -85,B 0,C 180,E1 -371.29,E2 -371.29} C_VEL
LIN {X 0,Y 608.53,Z 639.767,A -85,B 0,C 180,E1 -371.639,E2 -371.639} C_VEL
LIN {X 0,Y 608.559,Z 627.504,A -85,B 0,C 180,E1 -371.85,E2 -371.85} C_VEL
LIN {X 0,Y 608.466,Z 524.615,A -85,B 0,C 180,E1 -373.08,E2 -373.08} C_VEL
LIN {X 0,Y 608.495,Z 503.661,A -85,B 0,C 180,E1 -375.749,E2 -375.749} C_VEL
LIN {X 0,Y 608.539,Z 482.36,A -85,B 0,C 180,E1 -378.497,E2 -378.497} C_VEL
LIN {X 0,Y 608.561,Z 460.746,A -85,B 0,C 180,E1 -381.332,E2 -381.332} C_VEL
LIN {X 0,Y 608.45,Z 446.328,A -85,B 0,C 180,E1 -383.259,E2 -383.259} C_VEL
LIN {X 0,Y 608.456,Z 446.318,A -85,B 0,C 180,E1 -386.035,E2 -386.035} C_VEL
LIN {X 0,Y 608.479,Z 446.314,A -85,B 0,C 180,E1 -388.62,E2 -388.62} C_VEL
LIN {X 0,Y 608.448,Z 446.313,A -85,B 0,C 180,E1 -391.318,E2 -391.318} C_VEL
LIN {X 0,Y 608.476,Z 446.314,A -85,B 0,C 180,E1 -393.735,E2 -393.735} C_VEL
LIN {X 0,Y 608.482,Z 446.319,A -85,B 0,C 180,E1 -396.09,E2 -396.09} C_VEL
LIN {X 0,Y 608.47,Z 446.312,A -85,B 0,C 180,E1 -398.588,E2 -398.588} C_VEL
LIN {X 0,Y 608.457,Z 446.314,A -85,B 0,C 180,E1 -401.341,E2 -401.341} C_VEL
LIN {X 0,Y 608.45,Z 446.317,A -85,B 0,C 180,E1 -404.263,E2 -404.263} C_VEL
LIN {X 0,Y 608.454,Z 446.313,A -85,B 0,C 180,E1 -407.04,E2 -407.04} C_VEL
LIN {X 0,Y 608.457,Z 446.323,A -85,B 0,C 180,E1 -409.696,E2 -409.696} C_VEL
LIN {X 0,Y 608.471,Z 446.312,A -85,B 0,C 180,E1 -412.253,E2 -412.253} C_VEL
LIN {X 0,Y 608.451,Z 446.316,A -85,B 0,C 180,E1 -415.094,E2 -415.094} C_VEL
LIN {X 0,Y 608.47,Z 446.314,A -85,B 0,C 180,E1 -417.905,E2 -417.905} C_VEL
LIN {X 0,Y 608.461,Z 446.312,A -85,B 0,C 180,E1 -420.219,E2 -420.219} C_VEL
LIN {X 0,Y 608.484,Z 446.311,A -85,B 0,C 180,E1 -422.792,E2 -422.792} C_VEL
LIN {X 0,Y 608.484,Z 446.312,A -85,B 0,C 180,E1 -425.846,E2 -425.846} C_VEL
LIN {X 0,Y 608.499,Z 446.453,A -85,B 0,C 180,E1 -426.224,E2 -426.224} C_VEL
LIN {X 0,Y 608.652,Z 461.065,A -85,B 0,C 180,E1 -427.78,E2 -427.78} C_VEL
LIN {X 0,Y 608.584,Z 486.477,A -85,B 0,C 180,E1 -430.433,E2 -430.433} C_VEL
LIN {X 0,Y 608.546,Z 515.829,A -85,B 0,C 180,E1 -433.447,E2 -433.447} C_VEL
LIN {X 0,Y 608.549,Z 523.326,A -85,B 0,C 180,E1 -434.209,E2 -434.209} C_VEL
LIN {X 0,Y 608.615,Z 662.941,A -85,B 0,C 180,E1 -435.903,E2 -435.903} C_VEL
LIN {X 0,Y 608.583,Z 676.597,A -85,B 0,C 180,E1 -436.199,E2 -436.199} C_VEL
LIN {X 0,Y 608.581,Z 690.69,A -85,B 0,C 180,E1 -436.645,E2 -436.645} C_VEL
LIN {X 0,Y 608.562,Z 702.866,A -85,B 0,C 180,E1 -437.155,E2 -437.155} C_VEL
LIN {X 0,Y 608.516,Z 715.667,A -85,B 0,C 180,E1 -437.831,E2 -437.831} C_VEL
LIN {X 0,Y 608.499,Z 728.459,A -85,B 0,C 180,E1 -438.676,E2 -438.676} C_VEL
LIN {X 0,Y 608.496,Z 738.922,A -85,B 0,C 180,E1 -439.518,E2 -439.518} C_VEL
LIN {X 0,Y 608.479,Z 749.326,A -85,B 0,C 180,E1 -440.526,E2 -440.526} C_VEL
LIN {X 0,Y 608.464,Z 757.907,A -85,B 0,C 180,E1 -441.531,E2 -441.531} C_VEL
LIN {X 0,Y 608.461,Z 766.108,A -85,B 0,C 180,E1 -442.7,E2 -442.7} C_VEL
LIN {X 0,Y 608.443,Z 772.544,A -85,B 0,C 180,E1 -443.83,E2 -443.83} C_VEL
LIN {X 0,Y 608.437,Z 777.959,A -85,B 0,C 180,E1 -445.029,E2 -445.029} C_VEL
LIN {X 0,Y 608.432,Z 781.439,A -85,B 0,C 180,E1 -446.025,E2 -446.025} C_VEL
LIN {X 0,Y 608.424,Z 784.829,A -85,B 0,C 180,E1 -447.351,E2 -447.351} C_VEL
LIN {X 0,Y 608.442,Z 786.829,A -85,B 0,C 180,E1 -448.675,E2 -448.675} C_VEL
LIN {X 0,Y 608.433,Z 787.5,A -85,B 0,C 180,E1 -449.999,E2 -449.999} C_VEL
LIN {X 0,Y 608.442,Z 786.831,A -85,B 0,C 180,E1 -451.323,E2 -451.323} C_VEL
LIN {X 0,Y 608.424,Z 784.833,A -85,B 0,C 180,E1 -452.647,E2 -452.647} C_VEL
LIN {X 0,Y 608.431,Z 781.444,A -85,B 0,C 180,E1 -453.973,E2 -453.973} C_VEL
LIN {X 0,Y 608.44,Z 776.571,A -85,B 0,C 180,E1 -455.301,E2 -455.301} C_VEL
LIN {X 0,Y 608.444,Z 770.216,A -85,B 0,C 180,E1 -456.603,E2 -456.603} C_VEL
LIN {X 0,Y 608.453,Z 762.804,A -85,B 0,C 180,E1 -457.799,E2 -457.799} C_VEL
LIN {X 0,Y 608.472,Z 753.831,A -85,B 0,C 180,E1 -458.97,E2 -458.97} C_VEL
LIN {X 0,Y 608.472,Z 744.401,A -85,B 0,C 180,E1 -459.976,E2 -459.976} C_VEL
LIN {X 0,Y 608.505,Z 733.051,A -85,B 0,C 180,E1 -460.973,E2 -460.973} C_VEL
LIN {X 0,Y 608.532,Z 721.162,A -85,B 0,C 180,E1 -461.828,E2 -461.828} C_VEL
LIN {X 0,Y 608.531,Z 708.09,A -85,B 0,C 180,E1 -462.59,E2 -462.59} C_VEL
LIN {X 0,Y 608.562,Z 695.196,A -85,B 0,C 180,E1 -463.183,E2 -463.183} C_VEL
LIN {X 0,Y 608.585,Z 681.216,A -85,B 0,C 180,E1 -463.672,E2 -463.672} C_VEL
LIN {X 0,Y 608.596,Z 667.505,A -85,B 0,C 180,E1 -464.012,E2 -464.012} C_VEL
LIN {X 0,Y 608.622,Z 651.246,A -85,B 0,C 180,E1 -464.256,E2 -464.256} C_VEL
LIN {X 0,Y 608.549,Z 523.343,A -85,B 0,C 180,E1 -465.789,E2 -465.789} C_VEL
LIN {X 0,Y 608.565,Z 495.714,A -85,B 0,C 180,E1 -468.613,E2 -468.613} C_VEL
LIN {X 0,Y 608.641,Z 469.553,A -85,B 0,C 180,E1 -471.328,E2 -471.328} C_VEL
LIN {X 0,Y 608.671,Z 447.529,A -85,B 0,C 180,E1 -473.655,E2 -473.655} C_VEL
LIN {X 0,Y 608.452,Z 446.314,A -85,B 0,C 180,E1 -473.799,E2 -473.799} C_VEL
LIN {X 0,Y 608.459,Z 446.322,A -85,B 0,C 180,E1 -476.773,E2 -476.773} C_VEL
LIN {X 0,Y 608.47,Z 446.316,A -85,B 0,C 180,E1 -479.018,E2 -479.018} C_VEL
LIN {X 0,Y 608.474,Z 446.311,A -85,B 0,C 180,E1 -481.315,E2 -481.315} C_VEL
LIN {X 0,Y 608.468,Z 446.31,A -85,B 0,C 180,E1 -483.734,E2 -483.734} C_VEL
LIN {X 0,Y 608.473,Z 446.311,A -85,B 0,C 180,E1 -486.089,E2 -486.089} C_VEL
LIN {X 0,Y 608.472,Z 446.319,A -85,B 0,C 180,E1 -488.586,E2 -488.586} C_VEL
LIN {X 0,Y 608.461,Z 446.312,A -85,B 0,C 180,E1 -491.342,E2 -491.342} C_VEL
LIN {X 0,Y 608.46,Z 446.315,A -85,B 0,C 180,E1 -494.264,E2 -494.264} C_VEL
LIN {X 0,Y 608.455,Z 446.316,A -85,B 0,C 180,E1 -497.04,E2 -497.04} C_VEL
LIN {X 0,Y 608.446,Z 446.313,A -85,B 0,C 180,E1 -499.696,E2 -499.696} C_VEL
LIN {X 0,Y 608.466,Z 446.314,A -85,B 0,C 180,E1 -502.253,E2 -502.253} C_VEL
LIN {X 0,Y 608.483,Z 446.312,A -85,B 0,C 180,E1 -505.088,E2 -505.088} C_VEL
LIN {X 0,Y 608.463,Z 446.311,A -85,B 0,C 180,E1 -507.905,E2 -507.905} C_VEL
LIN {X 0,Y 608.472,Z 446.313,A -85,B 0,C 180,E1 -510.221,E2 -510.221} C_VEL
LIN {X 0,Y 608.479,Z 446.317,A -85,B 0,C 180,E1 -512.79,E2 -512.79} C_VEL
LIN {X 0,Y 608.448,Z 446.313,A -85,B 0,C 180,E1 -515.429,E2 -515.429} C_VEL
LIN {X 0,Y 608.471,Z 446.315,A -85,B 0,C 180,E1 -518.309,E2 -518.309} C_VEL
LIN {X 0,Y 608.469,Z 446.311,A -85,B 0,C 180,E1 -521.28,E2 -521.28} C_VEL
LIN {X 0,Y 608.456,Z 446.313,A -85,B 0,C 180,E1 -523.906,E2 -523.906} C_VEL
LIN {X 0,Y 608.463,Z 446.321,A -85,B 0,C 180,E1 -526.644,E2 -526.644} C_VEL
LIN {X 0,Y 608.465,Z 446.311,A -85,B 0,C 180,E1 -529.35,E2 -529.35} C_VEL
LIN {X 0,Y 608.47,Z 446.312,A -85,B 0,C 180,E1 -532.033,E2 -532.033} C_VEL
LIN {X 0,Y 608.466,Z 446.319,A -85,B 0,C 180,E1 -534.698,E2 -534.698} C_VEL
LIN {X 0,Y 608.481,Z 446.309,A -85,B 0,C 180,E1 -537.352,E2 -537.352} C_VEL
LIN {X 0,Y 608.467,Z 446.312,A -85,B 0,C 180,E1 -540,E2 -540} C_VEL
LIN {X 0,Y 608.484,Z 446.318,A -85,B 0,C 180,E1 -542.648,E2 -542.648} C_VEL
LIN {X 0,Y 608.457,Z 446.312,A -85,B 0,C 180,E1 -545.302,E2 -545.302} C_VEL
LIN {X 0,Y 608.471,Z 446.312,A -85,B 0,C 180,E1 -547.967,E2 -547.967} C_VEL
LIN {X 0,Y 608.451,Z 446.312,A -85,B 0,C 180,E1 -549.473,E2 -549.473} C_VEL
LIN {X 0,Y 607.773,Z 446.4,A -85,B 0,C 180,E1 -550.025,E2 -550.025} C_VEL
LIN {X 0,Y 604.92,Z 446.757,A -85,B 0,C 180,E1 -550.922,E2 -550.922} C_VEL
LIN {X 0,Y 602.517,Z 447.056,A -85,B 0,C 180,E1 -551.644,E2 -551.644} C_VEL
LIN {X 0,Y 601.489,Z 447.184,A -85,B 0,C 180,E1 -552.201,E2 -552.201} C_VEL
LIN {X 0,Y 601.406,Z 447.193,A -85,B 0,C 180,E1 -552.389,E2 -552.389} C_VEL
LIN {X 0,Y 601.426,Z 447.192,A -85,B 0,C 180,E1 -554.897,E2 -554.897} C_VEL
LIN {X 0,Y 601.426,Z 447.191,A -85,B 0,C 180,E1 -556.986,E2 -556.986} C_VEL
LIN {X 0,Y 601.402,Z 447.191,A -85,B 0,C 180,E1 -559.81,E2 -559.81} C_VEL
LIN {X 0,Y 601.408,Z 447.199,A -85,B 0,C 180,E1 -562.607,E2 -562.607} C_VEL
LIN {X 0,Y 601.399,Z 447.195,A -85,B 0,C 180,E1 -564.879,E2 -564.879} C_VEL
LIN {X 0,Y 601.419,Z 447.19,A -85,B 0,C 180,E1 -567.868,E2 -567.868} C_VEL
LIN {X 0,Y 601.44,Z 447.19,A -85,B 0,C 180,E1 -570.164,E2 -570.164} C_VEL
LIN {X 0,Y 601.421,Z 447.195,A -85,B 0,C 180,E1 -572.718,E2 -572.718} C_VEL
LIN {X 0,Y 601.415,Z 447.19,A -85,B 0,C 180,E1 -575.117,E2 -575.117} C_VEL
LIN {X 0,Y 601.428,Z 447.187,A -85,B 0,C 180,E1 -577.42,E2 -577.42} C_VEL
LIN {X 0,Y 601.411,Z 447.192,A -85,B 0,C 180,E1 -579.995,E2 -579.995} C_VEL
LIN {X 0,Y 601.407,Z 447.197,A -85,B 0,C 180,E1 -582.671,E2 -582.671} C_VEL
LIN {X 0,Y 601.42,Z 447.188,A -85,B 0,C 180,E1 -585.483,E2 -585.483} C_VEL
LIN {X 0,Y 601.427,Z 447.197,A -85,B 0,C 180,E1 -588.407,E2 -588.407} C_VEL
LIN {X 0,Y 601.434,Z 447.19,A -85,B 0,C 180,E1 -590.877,E2 -590.877} C_VEL
LIN {X 0,Y 601.441,Z 447.186,A -85,B 0,C 180,E1 -593.735,E2 -593.735} C_VEL
LIN {X 0,Y 601.431,Z 447.193,A -85,B 0,C 180,E1 -596.688,E2 -596.688} C_VEL
LIN {X 0,Y 601.431,Z 447.189,A -85,B 0,C 180,E1 -599.06,E2 -599.06} C_VEL
LIN {X 0,Y 601.427,Z 447.188,A -85,B 0,C 180,E1 -601.374,E2 -601.374} C_VEL
LIN {X 0,Y 601.404,Z 447.191,A -85,B 0,C 180,E1 -603.638,E2 -603.638} C_VEL
LIN {X 0,Y 601.423,Z 447.198,A -85,B 0,C 180,E1 -606.591,E2 -606.591} C_VEL
LIN {X 0,Y 601.448,Z 447.307,A -85,B 0,C 180,E1 -607.455,E2 -607.455} C_VEL
LIN {X 0,Y 601.65,Z 456.537,A -85,B 0,C 180,E1 -608.771,E2 -608.771} C_VEL
LIN {X 0,Y 601.569,Z 475.192,A -85,B 0,C 180,E1 -611.378,E2 -611.378} C_VEL
LIN {X 0,Y 601.484,Z 494.702,A -85,B 0,C 180,E1 -614.064,E2 -614.064} C_VEL
LIN {X 0,Y 601.442,Z 513.786,A -85,B 0,C 180,E1 -616.658,E2 -616.658} C_VEL
LIN {X 0,Y 601.486,Z 515.558,A -85,B 0,C 180,E1 -616.874,E2 -616.874} C_VEL
LIN {X 0,Y 601.613,Z 623.379,A -85,B 0,C 180,E1 -618.183,E2 -618.183} C_VEL
LIN {X 0,Y 601.573,Z 636.669,A -85,B 0,C 180,E1 -618.482,E2 -618.482} C_VEL
LIN {X 0,Y 601.537,Z 649.082,A -85,B 0,C 180,E1 -618.896,E2 -618.896} C_VEL
LIN {X 0,Y 601.534,Z 660.268,A -85,B 0,C 180,E1 -619.397,E2 -619.397} C_VEL
LIN {X 0,Y 601.482,Z 672.037,A -85,B 0,C 180,E1 -620.077,E2 -620.077} C_VEL
LIN {X 0,Y 601.444,Z 682.544,A -85,B 0,C 180,E1 -620.84,E2 -620.84} C_VEL
LIN {X 0,Y 601.429,Z 691.15,A -85,B 0,C 180,E1 -621.602,E2 -621.602} C_VEL
LIN {X 0,Y 601.417,Z 699.077,A -85,B 0,C 180,E1 -622.447,E2 -622.447} C_VEL
LIN {X 0,Y 601.376,Z 706.394,A -85,B 0,C 180,E1 -623.394,E2 -623.394} C_VEL
LIN {X 0,Y 601.372,Z 712.118,A -85,B 0,C 180,E1 -624.3,E2 -624.3} C_VEL
LIN {X 0,Y 601.335,Z 717.258,A -85,B 0,C 180,E1 -625.308,E2 -625.308} C_VEL
LIN {X 0,Y 601.367,Z 721.246,A -85,B 0,C 180,E1 -626.316,E2 -626.316} C_VEL
LIN {X 0,Y 601.324,Z 724.195,A -85,B 0,C 180,E1 -627.321,E2 -627.321} C_VEL
LIN {X 0,Y 601.342,Z 725.629,A -85,B 0,C 180,E1 -627.992,E2 -627.992} C_VEL
LIN {X 0,Y 601.339,Z 727.253,A -85,B 0,C 180,E1 -629.331,E2 -629.331} C_VEL
LIN {X 0,Y 601.336,Z 727.496,A -85,B 0,C 180,E1 -630.001,E2 -630.001} C_VEL
LIN {X 0,Y 601.339,Z 727.314,A -85,B 0,C 180,E1 -630.671,E2 -630.671} C_VEL
LIN {X 0,Y 601.343,Z 725.774,A -85,B 0,C 180,E1 -632.01,E2 -632.01} C_VEL
LIN {X 0,Y 601.326,Z 724.415,A -85,B 0,C 180,E1 -632.68,E2 -632.68} C_VEL
LIN {X 0,Y 601.368,Z 721.537,A -85,B 0,C 180,E1 -633.686,E2 -633.686} C_VEL
LIN {X 0,Y 601.337,Z 717.637,A -85,B 0,C 180,E1 -634.694,E2 -634.694} C_VEL
LIN {X 0,Y 601.373,Z 712.605,A -85,B 0,C 180,E1 -635.702,E2 -635.702} C_VEL
LIN {X 0,Y 601.383,Z 706.286,A -85,B 0,C 180,E1 -636.712,E2 -636.712} C_VEL
LIN {X 0,Y 601.397,Z 698.367,A -85,B 0,C 180,E1 -637.724,E2 -637.724} C_VEL
LIN {X 0,Y 601.437,Z 688.521,A -85,B 0,C 180,E1 -638.738,E2 -638.738} C_VEL
LIN {X 0,Y 601.449,Z 678.197,A -85,B 0,C 180,E1 -639.586,E2 -639.586} C_VEL
LIN {X 0,Y 601.492,Z 666.576,A -85,B 0,C 180,E1 -640.35,E2 -640.35} C_VEL
LIN {X 0,Y 601.551,Z 655.356,A -85,B 0,C 180,E1 -640.929,E2 -640.929} C_VEL
LIN {X 0,Y 601.557,Z 642.801,A -85,B 0,C 180,E1 -641.421,E2 -641.421} C_VEL
LIN {X 0,Y 601.587,Z 630.003,A -85,B 0,C 180,E1 -641.776,E2 -641.776} C_VEL
LIN {X 0,Y 601.6,Z 617.694,A -85,B 0,C 180,E1 -641.99,E2 -641.99} C_VEL
LIN {X 0,Y 601.642,Z 516.642,A -85,B 0,C 180,E1 -643.2,E2 -643.2} C_VEL
LIN {X 0,Y 601.468,Z 515.075,A -85,B 0,C 180,E1 -643.257,E2 -643.257} C_VEL
LIN {X 0,Y 601.498,Z 494.074,A -85,B 0,C 180,E1 -646.112,E2 -646.112} C_VEL
LIN {X 0,Y 601.565,Z 475.837,A -85,B 0,C 180,E1 -648.622,E2 -648.622} C_VEL
LIN {X 0,Y 601.664,Z 454.616,A -85,B 0,C 180,E1 -651.59,E2 -651.59} C_VEL
LIN {X 0,Y 601.418,Z 447.202,A -85,B 0,C 180,E1 -652.652,E2 -652.652} C_VEL
LIN {X 0,Y 601.407,Z 447.191,A -85,B 0,C 180,E1 -654.879,E2 -654.879} C_VEL
LIN {X 0,Y 601.425,Z 447.196,A -85,B 0,C 180,E1 -657.868,E2 -657.868} C_VEL
LIN {X 0,Y 601.435,Z 447.19,A -85,B 0,C 180,E1 -660.164,E2 -660.164} C_VEL
LIN {X 0,Y 601.422,Z 447.188,A -85,B 0,C 180,E1 -662.715,E2 -662.715} C_VEL
LIN {X 0,Y 601.398,Z 447.193,A -85,B 0,C 180,E1 -665.112,E2 -665.112} C_VEL
LIN {X 0,Y 601.441,Z 447.192,A -85,B 0,C 180,E1 -667.419,E2 -667.419} C_VEL
LIN {X 0,Y 601.417,Z 447.194,A -85,B 0,C 180,E1 -669.995,E2 -669.995} C_VEL
LIN {X 0,Y 601.416,Z 447.189,A -85,B 0,C 180,E1 -672.671,E2 -672.671} C_VEL
LIN {X 0,Y 601.432,Z 447.194,A -85,B 0,C 180,E1 -675.482,E2 -675.482} C_VEL
LIN {X 0,Y 601.425,Z 447.188,A -85,B 0,C 180,E1 -678.408,E2 -678.408} C_VEL
LIN {X 0,Y 601.415,Z 447.189,A -85,B 0,C 180,E1 -680.873,E2 -680.873} C_VEL
LIN {X 0,Y 601.448,Z 447.195,A -85,B 0,C 180,E1 -683.734,E2 -683.734} C_VEL
LIN {X 0,Y 601.431,Z 447.187,A -85,B 0,C 180,E1 -686.686,E2 -686.686} C_VEL
LIN {X 0,Y 601.417,Z 447.19,A -85,B 0,C 180,E1 -689.058,E2 -689.058} C_VEL
LIN {X 0,Y 601.439,Z 447.191,A -85,B 0,C 180,E1 -691.373,E2 -691.373} C_VEL
LIN {X 0,Y 601.421,Z 447.192,A -85,B 0,C 180,E1 -694.132,E2 -694.132} C_VEL
LIN {X 0,Y 601.468,Z 447.337,A -85,B 0,C 180,E1 -696.683,E2 -696.683} C_VEL
LIN {X 0,Y 601.718,Z 452.894,A -85,B 0,C 180,E1 -697.446,E2 -697.446} C_VEL
LIN {X 0,Y 601.629,Z 474.813,A -85,B 0,C 180,E1 -700.376,E2 -700.376} C_VEL
LIN {X 0,Y 601.55,Z 496.174,A -85,B 0,C 180,E1 -703.181,E2 -703.181} C_VEL
LIN {X 0,Y 601.485,Z 518.097,A -85,B 0,C 180,E1 -706.019,E2 -706.019} C_VEL
LIN {X 0,Y 601.459,Z 524.577,A -85,B 0,C 180,E1 -706.85,E2 -706.85} C_VEL
LIN {X 0,Y 601.674,Z 530.535,A -85,B 0,C 180,E1 -706.941,E2 -706.941} C_VEL
LIN {X 0,Y 601.627,Z 632.969,A -85,B 0,C 180,E1 -708.182,E2 -708.182} C_VEL
LIN {X 0,Y 601.581,Z 646.353,A -85,B 0,C 180,E1 -708.481,E2 -708.481} C_VEL
LIN {X 0,Y 601.552,Z 659.627,A -85,B 0,C 180,E1 -708.928,E2 -708.928} C_VEL
LIN {X 0,Y 601.507,Z 671.576,A -85,B 0,C 180,E1 -709.481,E2 -709.481} C_VEL
LIN {X 0,Y 601.47,Z 683.004,A -85,B 0,C 180,E1 -710.16,E2 -710.16} C_VEL
LIN {X 0,Y 601.438,Z 693.299,A -85,B 0,C 180,E1 -710.923,E2 -710.923} C_VEL
LIN {X 0,Y 601.411,Z 702.562,A -85,B 0,C 180,E1 -711.77,E2 -711.77} C_VEL
LIN {X 0,Y 601.389,Z 711.534,A -85,B 0,C 180,E1 -712.783,E2 -712.783} C_VEL
LIN {X 0,Y 601.376,Z 718.67,A -85,B 0,C 180,E1 -713.781,E2 -713.781} C_VEL
LIN {X 0,Y 601.373,Z 723.64,A -85,B 0,C 180,E1 -714.635,E2 -714.635} C_VEL
LIN {X 0,Y 601.353,Z 728.383,A -85,B 0,C 180,E1 -715.643,E2 -715.643} C_VEL
LIN {X 0,Y 601.345,Z 732.02,A -85,B 0,C 180,E1 -716.65,E2 -716.65} C_VEL
LIN {X 0,Y 601.324,Z 733.903,A -85,B 0,C 180,E1 -717.32,E2 -717.32} C_VEL
LIN {X 0,Y 601.341,Z 735.338,A -85,B 0,C 180,E1 -717.991,E2 -717.991} C_VEL
LIN {X 0,Y 601.339,Z 736.963,A -85,B 0,C 180,E1 -719.33,E2 -719.33} C_VEL
LIN {X 0,Y 601.335,Z 737.206,A -85,B 0,C 180,E1 -720,E2 -720} C_VEL
LIN {X 0,Y 601.339,Z 737.026,A -85,B 0,C 180,E1 -720.67,E2 -720.67} C_VEL
LIN {X 0,Y 601.34,Z 735.487,A -85,B 0,C 180,E1 -722.009,E2 -722.009} C_VEL
LIN {X 0,Y 601.326,Z 734.119,A -85,B 0,C 180,E1 -722.679,E2 -722.679} C_VEL
LIN {X 0,Y 601.368,Z 731.244,A -85,B 0,C 180,E1 -723.685,E2 -723.685} C_VEL
LIN {X 0,Y 601.337,Z 727.343,A -85,B 0,C 180,E1 -724.693,E2 -724.693} C_VEL
LIN {X 0,Y 601.373,Z 722.314,A -85,B 0,C 180,E1 -725.701,E2 -725.701} C_VEL
LIN {X 0,Y 601.383,Z 716.001,A -85,B 0,C 180,E1 -726.711,E2 -726.711} C_VEL
LIN {X 0,Y 601.396,Z 708.086,A -85,B 0,C 180,E1 -727.723,E2 -727.723} C_VEL
LIN {X 0,Y 601.422,Z 700.02,A -85,B 0,C 180,E1 -728.568,E2 -728.568} C_VEL
LIN {X 0,Y 601.453,Z 690.18,A -85,B 0,C 180,E1 -729.415,E2 -729.415} C_VEL
LIN {X 0,Y 601.478,Z 679.129,A -85,B 0,C 180,E1 -730.179,E2 -730.179} C_VEL
LIN {X 0,Y 601.532,Z 666.734,A -85,B 0,C 180,E1 -730.851,E2 -730.851} C_VEL
LIN {X 0,Y 601.553,Z 654.933,A -85,B 0,C 180,E1 -731.339,E2 -731.339} C_VEL
LIN {X 0,Y 601.574,Z 642.479,A -85,B 0,C 180,E1 -731.712,E2 -731.712} C_VEL
LIN {X 0,Y 601.618,Z 628.973,A -85,B 0,C 180,E1 -731.967,E2 -731.967} C_VEL
LIN {X 0,Y 601.561,Z 525.526,A -85,B 0,C 180,E1 -733.212,E2 -733.212} C_VEL
LIN {X 0,Y 601.452,Z 524.611,A -85,B 0,C 180,E1 -733.235,E2 -733.235} C_VEL
LIN {X 0,Y 601.524,Z 503.657,A -85,B 0,C 180,E1 -735.936,E2 -735.936} C_VEL
LIN {X 0,Y 601.582,Z 481.259,A -85,B 0,C 180,E1 -738.864,E2 -738.864} C_VEL
LIN {X 0,Y 601.679,Z 459.4,A -85,B 0,C 180,E1 -741.769,E2 -741.769} C_VEL
LIN {X 0,Y 601.694,Z 448.671,A -85,B 0,C 180,E1 -743.217,E2 -743.217} C_VEL
LIN {X 0,Y 601.429,Z 447.192,A -85,B 0,C 180,E1 -743.456,E2 -743.456} C_VEL
LIN {X 0,Y 601.408,Z 447.2,A -85,B 0,C 180,E1 -746.363,E2 -746.363} C_VEL
LIN {X 0,Y 601.443,Z 447.188,A -85,B 0,C 180,E1 -748.789,E2 -748.789} C_VEL
LIN {X 0,Y 601.424,Z 447.19,A -85,B 0,C 180,E1 -751.454,E2 -751.454} C_VEL
LIN {X 0,Y 601.435,Z 447.197,A -85,B 0,C 180,E1 -754.118,E2 -754.118} C_VEL
LIN {X 0,Y 601.412,Z 447.192,A -85,B 0,C 180,E1 -756.582,E2 -756.582} C_VEL
LIN {X 0,Y 601.416,Z 447.19,A -85,B 0,C 180,E1 -759.126,E2 -759.126} C_VEL
LIN {X 0,Y 601.426,Z 447.196,A -85,B 0,C 180,E1 -761.765,E2 -761.765} C_VEL
LIN {X 0,Y 601.401,Z 447.192,A -85,B 0,C 180,E1 -764.532,E2 -764.532} C_VEL
LIN {X 0,Y 601.455,Z 447.186,A -85,B 0,C 180,E1 -766.425,E2 -766.425} C_VEL
LIN {X 0,Y 601.417,Z 447.195,A -85,B 0,C 180,E1 -769.427,E2 -769.427} C_VEL
LIN {X 0,Y 601.424,Z 447.197,A -85,B 0,C 180,E1 -771.732,E2 -771.732} C_VEL
LIN {X 0,Y 601.388,Z 447.194,A -85,B 0,C 180,E1 -774.245,E2 -774.245} C_VEL
LIN {X 0,Y 601.421,Z 447.189,A -85,B 0,C 180,E1 -776.685,E2 -776.685} C_VEL
LIN {X 0,Y 601.42,Z 447.193,A -85,B 0,C 180,E1 -779.057,E2 -779.057} C_VEL
LIN {X 0,Y 601.438,Z 447.197,A -85,B 0,C 180,E1 -781.373,E2 -781.373} C_VEL
LIN {X 0,Y 601.406,Z 447.197,A -85,B 0,C 180,E1 -783.636,E2 -783.636} C_VEL
LIN {X 0,Y 601.457,Z 447.3,A -85,B 0,C 180,E1 -786.019,E2 -786.019} C_VEL
LIN {X 0,Y 601.863,Z 450.9,A -85,B 0,C 180,E1 -786.425,E2 -786.425} C_VEL
LIN {X 0,Y 601.759,Z 476.202,A -85,B 0,C 180,E1 -789.12,E2 -789.12} C_VEL
LIN {X 0,Y 601.638,Z 501.725,A -85,B 0,C 180,E1 -791.791,E2 -791.791} C_VEL
LIN {X 0,Y 601.568,Z 523.326,A -85,B 0,C 180,E1 -794.021,E2 -794.021} C_VEL
LIN {X 0,Y 601.843,Z 528.553,A -85,B 0,C 180,E1 -794.094,E2 -794.094} C_VEL
LIN {X 0,Y 601.721,Z 662.941,A -85,B 0,C 180,E1 -795.738,E2 -795.738} C_VEL
LIN {X 0,Y 601.693,Z 677.049,A -85,B 0,C 180,E1 -796.05,E2 -796.05} C_VEL
LIN {X 0,Y 601.667,Z 690.691,A -85,B 0,C 180,E1 -796.489,E2 -796.489} C_VEL
LIN {X 0,Y 601.607,Z 704.617,A -85,B 0,C 180,E1 -797.089,E2 -797.089} C_VEL
LIN {X 0,Y 601.546,Z 717.08,A -85,B 0,C 180,E1 -797.774,E2 -797.774} C_VEL
LIN {X 0,Y 601.505,Z 728.461,A -85,B 0,C 180,E1 -798.542,E2 -798.542} C_VEL
LIN {X 0,Y 601.482,Z 738.923,A -85,B 0,C 180,E1 -799.395,E2 -799.395} C_VEL
LIN {X 0,Y 601.43,Z 749.326,A -85,B 0,C 180,E1 -800.414,E2 -800.414} C_VEL
LIN {X 0,Y 601.407,Z 757.907,A -85,B 0,C 180,E1 -801.43,E2 -801.43} C_VEL
LIN {X 0,Y 601.392,Z 766.109,A -85,B 0,C 180,E1 -802.613,E2 -802.613} C_VEL
LIN {X 0,Y 601.361,Z 771.751,A -85,B 0,C 180,E1 -803.604,E2 -803.604} C_VEL
LIN {X 0,Y 601.355,Z 776.564,A -85,B 0,C 180,E1 -804.634,E2 -804.634} C_VEL
LIN {X 0,Y 601.343,Z 781.439,A -85,B 0,C 180,E1 -805.978,E2 -805.978} C_VEL
LIN {X 0,Y 601.323,Z 784.829,A -85,B 0,C 180,E1 -807.32,E2 -807.32} C_VEL
LIN {X 0,Y 601.342,Z 786.83,A -85,B 0,C 180,E1 -808.66,E2 -808.66} C_VEL
LIN {X 0,Y 601.333,Z 787.5,A -85,B 0,C 180,E1 -809.999,E2 -809.999} C_VEL
LIN {X 0,Y 601.342,Z 786.832,A -85,B 0,C 180,E1 -811.338,E2 -811.338} C_VEL
LIN {X 0,Y 601.323,Z 784.833,A -85,B 0,C 180,E1 -812.679,E2 -812.679} C_VEL
LIN {X 0,Y 601.343,Z 781.445,A -85,B 0,C 180,E1 -814.02,E2 -814.02} C_VEL
LIN {X 0,Y 601.354,Z 776.571,A -85,B 0,C 180,E1 -815.364,E2 -815.364} C_VEL
LIN {X 0,Y 601.371,Z 770.626,A -85,B 0,C 180,E1 -816.604,E2 -816.604} C_VEL
LIN {X 0,Y 601.385,Z 763.925,A -85,B 0,C 180,E1 -817.723,E2 -817.723} C_VEL
LIN {X 0,Y 601.411,Z 755.206,A -85,B 0,C 180,E1 -818.906,E2 -818.906} C_VEL
LIN {X 0,Y 601.432,Z 746.091,A -85,B 0,C 180,E1 -819.924,E2 -819.924} C_VEL
LIN {X 0,Y 601.496,Z 735.831,A -85,B 0,C 180,E1 -820.876,E2 -820.876} C_VEL
LIN {X 0,Y 601.533,Z 724.984,A -85,B 0,C 180,E1 -821.711,E2 -821.711} C_VEL
LIN {X 0,Y 601.575,Z 712.794,A -85,B 0,C 180,E1 -822.481,E2 -822.481} C_VEL
LIN {X 0,Y 601.629,Z 701.115,A -85,B 0,C 180,E1 -823.08,E2 -823.08} C_VEL
LIN {X 0,Y 601.651,Z 688.961,A -85,B 0,C 180,E1 -823.577,E2 -823.577} C_VEL
LIN {X 0,Y 601.683,Z 675.045,A -85,B 0,C 180,E1 -824.005,E2 -824.005} C_VEL
LIN {X 0,Y 601.74,Z 660.97,A -85,B 0,C 180,E1 -824.294,E2 -824.294} C_VEL
LIN {X 0,Y 601.728,Z 524.343,A -85,B 0,C 180,E1 -825.961,E2 -825.961} C_VEL
LIN {X 0,Y 601.567,Z 523.343,A -85,B 0,C 180,E1 -825.977,E2 -825.977} C_VEL
LIN {X 0,Y 601.645,Z 496.503,A -85,B 0,C 180,E1 -828.753,E2 -828.753} C_VEL
LIN {X 0,Y 601.777,Z 471.247,A -85,B 0,C 180,E1 -831.404,E2 -831.404} C_VEL
LIN {X 0,Y 601.848,Z 449.223,A -85,B 0,C 180,E1 -833.756,E2 -833.756} C_VEL
LIN {X 0,Y 601.452,Z 447.19,A -85,B 0,C 180,E1 -834.002,E2 -834.002} C_VEL
LIN {X 0,Y 601.456,Z 447.188,A -85,B 0,C 180,E1 -837.11,E2 -837.11} C_VEL
LIN {X 0,Y 601.415,Z 447.19,A -85,B 0,C 180,E1 -839.392,E2 -839.392} C_VEL
LIN {X 0,Y 601.413,Z 447.189,A -85,B 0,C 180,E1 -841.725,E2 -841.725} C_VEL
LIN {X 0,Y 601.428,Z 447.189,A -85,B 0,C 180,E1 -844.117,E2 -844.117} C_VEL
LIN {X 0,Y 601.414,Z 447.197,A -85,B 0,C 180,E1 -846.581,E2 -846.581} C_VEL
LIN {X 0,Y 601.436,Z 447.187,A -85,B 0,C 180,E1 -849.535,E2 -849.535} C_VEL
LIN {X 0,Y 601.436,Z 447.195,A -85,B 0,C 180,E1 -852.593,E2 -852.593} C_VEL
LIN {X 0,Y 601.418,Z 447.189,A -85,B 0,C 180,E1 -855.481,E2 -855.481} C_VEL
LIN {X 0,Y 601.424,Z 447.193,A -85,B 0,C 180,E1 -858.405,E2 -858.405} C_VEL
LIN {X 0,Y 601.435,Z 447.193,A -85,B 0,C 180,E1 -860.875,E2 -860.875} C_VEL
LIN {X 0,Y 601.437,Z 447.185,A -85,B 0,C 180,E1 -863.733,E2 -863.733} C_VEL
LIN {X 0,Y 601.432,Z 447.188,A -85,B 0,C 180,E1 -866.062,E2 -866.062} C_VEL
LIN {X 0,Y 601.436,Z 447.195,A -85,B 0,C 180,E1 -868.54,E2 -868.54} C_VEL
LIN {X 0,Y 601.431,Z 447.187,A -85,B 0,C 180,E1 -871.373,E2 -871.373} C_VEL
LIN {X 0,Y 601.415,Z 447.191,A -85,B 0,C 180,E1 -874.129,E2 -874.129} C_VEL
LIN {X 0,Y 601.419,Z 447.198,A -85,B 0,C 180,E1 -876.59,E2 -876.59} C_VEL
LIN {X 0,Y 601.428,Z 447.187,A -85,B 0,C 180,E1 -879.478,E2 -879.478} C_VEL
LIN {X 0,Y 601.397,Z 447.196,A -85,B 0,C 180,E1 -882.312,E2 -882.312} C_VEL
LIN {X 0,Y 601.428,Z 447.19,A -85,B 0,C 180,E1 -885.103,E2 -885.103} C_VEL
LIN {X 0,Y 601.414,Z 447.19,A -85,B 0,C 180,E1 -887.858,E2 -887.858} C_VEL
LIN {X 0,Y 601.416,Z 447.199,A -85,B 0,C 180,E1 -890.584,E2 -890.584} C_VEL
LIN {X 0,Y 601.444,Z 447.186,A -85,B 0,C 180,E1 -893.323,E2 -893.323} C_VEL
LIN {X 0,Y 601.399,Z 447.192,A -85,B 0,C 180,E1 -895.979,E2 -895.979} C_VEL
LIN {X 0,Y 601.427,Z 447.197,A -85,B 0,C 180,E1 -898.661,E2 -898.661} C_VEL
LIN {X 0,Y 601.422,Z 447.188,A -85,B 0,C 180,E1 -901.339,E2 -901.339} C_VEL
LIN {X 0,Y 601.427,Z 447.187,A -85,B 0,C 180,E1 -903.35,E2 -903.35} C_VEL
LIN {X 0,Y 601.406,Z 447.192,A -85,B 0,C 180,E1 -906.037,E2 -906.037} C_VEL
LIN {X 0,Y 601.435,Z 447.194,A -85,B 0,C 180,E1 -908.738,E2 -908.738} C_VEL
LIN {X 0,Y 601.426,Z 447.187,A -85,B 0,C 180,E1 -911.458,E2 -911.458} C_VEL
LIN {X 0,Y 601.406,Z 447.193,A -85,B 0,C 180,E1 -912.389,E2 -912.389} C_VEL
LIN {X 0,Y 600.743,Z 447.278,A -85,B 0,C 180,E1 -912.948,E2 -912.948} C_VEL
LIN {X 0,Y 597.891,Z 447.632,A -85,B 0,C 180,E1 -913.856,E2 -913.856} C_VEL
LIN {X 0,Y 595.479,Z 447.939,A -85,B 0,C 180,E1 -914.586,E2 -914.586} C_VEL
LIN {X 0,Y 594.441,Z 448.06,A -85,B 0,C 180,E1 -915.15,E2 -915.15} C_VEL
LIN {X 0,Y 594.356,Z 448.069,A -85,B 0,C 180,E1 -915.341,E2 -915.341} C_VEL
LIN {X 0,Y 594.374,Z 448.067,A -85,B 0,C 180,E1 -917.905,E2 -917.905} C_VEL
LIN {X 0,Y 594.377,Z 448.069,A -85,B 0,C 180,E1 -920.92,E2 -920.92} C_VEL
LIN {X 0,Y 594.386,Z 448.065,A -85,B 0,C 180,E1 -923.704,E2 -923.704} C_VEL
LIN {X 0,Y 594.381,Z 448.072,A -85,B 0,C 180,E1 -926.7,E2 -926.7} C_VEL
LIN {X 0,Y 594.38,Z 448.068,A -85,B 0,C 180,E1 -928.999,E2 -928.999} C_VEL
LIN {X 0,Y 594.386,Z 448.065,A -85,B 0,C 180,E1 -931.647,E2 -931.647} C_VEL
LIN {X 0,Y 594.393,Z 448.073,A -85,B 0,C 180,E1 -934.579,E2 -934.579} C_VEL
LIN {X 0,Y 594.379,Z 448.067,A -85,B 0,C 180,E1 -937.087,E2 -937.087} C_VEL
LIN {X 0,Y 594.375,Z 448.067,A -85,B 0,C 180,E1 -939.776,E2 -939.776} C_VEL
LIN {X 0,Y 594.365,Z 448.076,A -85,B 0,C 180,E1 -942.376,E2 -942.376} C_VEL
LIN {X 0,Y 594.357,Z 448.069,A -85,B 0,C 180,E1 -945.192,E2 -945.192} C_VEL
LIN {X 0,Y 594.369,Z 448.067,A -85,B 0,C 180,E1 -947.626,E2 -947.626} C_VEL
LIN {X 0,Y 594.391,Z 448.072,A -85,B 0,C 180,E1 -950.322,E2 -950.322} C_VEL
LIN {X 0,Y 594.384,Z 448.068,A -85,B 0,C 180,E1 -952.915,E2 -952.915} C_VEL
LIN {X 0,Y 594.383,Z 448.067,A -85,B 0,C 180,E1 -955.862,E2 -955.862} C_VEL
LIN {X 0,Y 594.391,Z 448.071,A -85,B 0,C 180,E1 -958.652,E2 -958.652} C_VEL
LIN {X 0,Y 594.381,Z 448.067,A -85,B 0,C 180,E1 -961.043,E2 -961.043} C_VEL
LIN {X 0,Y 594.39,Z 448.068,A -85,B 0,C 180,E1 -963.977,E2 -963.977} C_VEL
LIN {X 0,Y 594.394,Z 448.074,A -85,B 0,C 180,E1 -966.297,E2 -966.297} C_VEL
LIN {X 0,Y 594.391,Z 448.221,A -85,B 0,C 180,E1 -967.303,E2 -967.303} C_VEL
LIN {X 0,Y 594.731,Z 453.997,A -85,B 0,C 180,E1 -968.147,E2 -968.147} C_VEL
LIN {X 0,Y 594.602,Z 474.191,A -85,B 0,C 180,E1 -971.011,E2 -971.011} C_VEL
LIN {X 0,Y 594.51,Z 493.434,A -85,B 0,C 180,E1 -973.695,E2 -973.695} C_VEL
LIN {X 0,Y 594.437,Z 513.79,A -85,B 0,C 180,E1 -976.498,E2 -976.498} C_VEL
LIN {X 0,Y 594.464,Z 515.604,A -85,B 0,C 180,E1 -976.716,E2 -976.716} C_VEL
LIN {X 0,Y 594.75,Z 520.967,A -85,B 0,C 180,E1 -976.788,E2 -976.788} C_VEL
LIN {X 0,Y 594.666,Z 623.408,A -85,B 0,C 180,E1 -978.043,E2 -978.043} C_VEL
LIN {X 0,Y 594.615,Z 636.688,A -85,B 0,C 180,E1 -978.345,E2 -978.345} C_VEL
LIN {X 0,Y 594.553,Z 649.937,A -85,B 0,C 180,E1 -978.796,E2 -978.796} C_VEL
LIN {X 0,Y 594.514,Z 661.907,A -85,B 0,C 180,E1 -979.357,E2 -979.357} C_VEL
LIN {X 0,Y 594.472,Z 673.323,A -85,B 0,C 180,E1 -980.044,E2 -980.044} C_VEL
LIN {X 0,Y 594.406,Z 683.612,A -85,B 0,C 180,E1 -980.816,E2 -980.816} C_VEL
LIN {X 0,Y 594.373,Z 692.869,A -85,B 0,C 180,E1 -981.673,E2 -981.673} C_VEL
LIN {X 0,Y 594.316,Z 701.841,A -85,B 0,C 180,E1 -982.698,E2 -982.698} C_VEL
LIN {X 0,Y 594.285,Z 708.356,A -85,B 0,C 180,E1 -983.612,E2 -983.612} C_VEL
LIN {X 0,Y 594.289,Z 713.946,A -85,B 0,C 180,E1 -984.572,E2 -984.572} C_VEL
LIN {X 0,Y 594.27,Z 718.687,A -85,B 0,C 180,E1 -985.592,E2 -985.592} C_VEL
LIN {X 0,Y 594.267,Z 722.319,A -85,B 0,C 180,E1 -986.611,E2 -986.611} C_VEL
LIN {X 0,Y 594.225,Z 724.197,A -85,B 0,C 180,E1 -987.289,E2 -987.289} C_VEL
LIN {X 0,Y 594.241,Z 725.629,A -85,B 0,C 180,E1 -987.968,E2 -987.968} C_VEL
LIN {X 0,Y 594.24,Z 727.254,A -85,B 0,C 180,E1 -989.323,E2 -989.323} C_VEL
LIN {X 0,Y 594.236,Z 727.496,A -85,B 0,C 180,E1 -990.001,E2 -990.001} C_VEL
LIN {X 0,Y 594.239,Z 727.314,A -85,B 0,C 180,E1 -990.679,E2 -990.679} C_VEL
LIN {X 0,Y 594.242,Z 725.773,A -85,B 0,C 180,E1 -992.034,E2 -992.034} C_VEL
LIN {X 0,Y 594.226,Z 724.413,A -85,B 0,C 180,E1 -992.712,E2 -992.712} C_VEL
LIN {X 0,Y 594.289,Z 721.535,A -85,B 0,C 180,E1 -993.73,E2 -993.73} C_VEL
LIN {X 0,Y 594.242,Z 717.635,A -85,B 0,C 180,E1 -994.75,E2 -994.75} C_VEL
LIN {X 0,Y 594.299,Z 712.602,A -85,B 0,C 180,E1 -995.77,E2 -995.77} C_VEL
LIN {X 0,Y 594.317,Z 706.282,A -85,B 0,C 180,E1 -996.792,E2 -996.792} C_VEL
LIN {X 0,Y 594.347,Z 698.362,A -85,B 0,C 180,E1 -997.816,E2 -997.816} C_VEL
LIN {X 0,Y 594.382,Z 688.515,A -85,B 0,C 180,E1 -998.843,E2 -998.843} C_VEL
LIN {X 0,Y 594.431,Z 678.191,A -85,B 0,C 180,E1 -999.7,E2 -999.7} C_VEL
LIN {X 0,Y 594.508,Z 666.565,A -85,B 0,C 180,E1 -1000.473,E2 -1000.473} C_VEL
LIN {X 0,Y 594.565,Z 655.345,A -85,B 0,C 180,E1 -1001.059,E2 -1001.059} C_VEL
LIN {X 0,Y 594.593,Z 642.858,A -85,B 0,C 180,E1 -1001.554,E2 -1001.554} C_VEL
LIN {X 0,Y 594.643,Z 629.98,A -85,B 0,C 180,E1 -1001.916,E2 -1001.916} C_VEL
LIN {X 0,Y 594.679,Z 617.653,A -85,B 0,C 180,E1 -1002.131,E2 -1002.131} C_VEL
LIN {X 0,Y 594.662,Z 516.821,A -85,B 0,C 180,E1 -1003.355,E2 -1003.355} C_VEL
LIN {X 0,Y 594.412,Z 515.229,A -85,B 0,C 180,E1 -1003.396,E2 -1003.396} C_VEL
LIN {X 0,Y 594.507,Z 495.343,A -85,B 0,C 180,E1 -1006.13,E2 -1006.13} C_VEL
LIN {X 0,Y 594.581,Z 477.523,A -85,B 0,C 180,E1 -1008.612,E2 -1008.612} C_VEL
LIN {X 0,Y 594.721,Z 457.158,A -85,B 0,C 180,E1 -1011.491,E2 -1011.491} C_VEL
LIN {X 0,Y 594.722,Z 450.264,A -85,B 0,C 180,E1 -1012.479,E2 -1012.479} C_VEL
LIN {X 0,Y 594.367,Z 448.073,A -85,B 0,C 180,E1 -1012.813,E2 -1012.813} C_VEL
LIN {X 0,Y 594.382,Z 448.069,A -85,B 0,C 180,E1 -1015.194,E2 -1015.194} C_VEL
LIN {X 0,Y 594.393,Z 448.073,A -85,B 0,C 180,E1 -1017.527,E2 -1017.527} C_VEL
LIN {X 0,Y 594.393,Z 448.066,A -85,B 0,C 180,E1 -1020.329,E2 -1020.329} C_VEL
LIN {X 0,Y 594.384,Z 448.066,A -85,B 0,C 180,E1 -1022.951,E2 -1022.951} C_VEL
LIN {X 0,Y 594.356,Z 448.074,A -85,B 0,C 180,E1 -1025.409,E2 -1025.409} C_VEL
LIN {X 0,Y 594.393,Z 448.07,A -85,B 0,C 180,E1 -1027.941,E2 -1027.941} C_VEL
LIN {X 0,Y 594.381,Z 448.065,A -85,B 0,C 180,E1 -1030.822,E2 -1030.822} C_VEL
LIN {X 0,Y 594.389,Z 448.072,A -85,B 0,C 180,E1 -1033.841,E2 -1033.841} C_VEL
LIN {X 0,Y 594.371,Z 448.066,A -85,B 0,C 180,E1 -1036.701,E2 -1036.701} C_VEL
LIN {X 0,Y 594.375,Z 448.072,A -85,B 0,C 180,E1 -1039.433,E2 -1039.433} C_VEL
LIN {X 0,Y 594.393,Z 448.064,A -85,B 0,C 180,E1 -1042.392,E2 -1042.392} C_VEL
LIN {X 0,Y 594.389,Z 448.064,A -85,B 0,C 180,E1 -1044.672,E2 -1044.672} C_VEL
LIN {X 0,Y 594.384,Z 448.066,A -85,B 0,C 180,E1 -1047.088,E2 -1047.088} C_VEL
LIN {X 0,Y 594.391,Z 448.075,A -85,B 0,C 180,E1 -1049.672,E2 -1049.672} C_VEL
LIN {X 0,Y 594.38,Z 448.066,A -85,B 0,C 180,E1 -1052.539,E2 -1052.539} C_VEL
LIN {X 0,Y 594.38,Z 448.066,A -85,B 0,C 180,E1 -1054.807,E2 -1054.807} C_VEL
LIN {X 0,Y 594.401,Z 448.179,A -85,B 0,C 180,E1 -1056.504,E2 -1056.504} C_VEL
LIN {X 0,Y 594.83,Z 452.817,A -85,B 0,C 180,E1 -1057.159,E2 -1057.159} C_VEL
LIN {X 0,Y 594.688,Z 474.818,A -85,B 0,C 180,E1 -1060.137,E2 -1060.137} C_VEL
LIN {X 0,Y 594.573,Z 495.946,A -85,B 0,C 180,E1 -1062.947,E2 -1062.947} C_VEL
LIN {X 0,Y 594.45,Z 517.756,A -85,B 0,C 180,E1 -1065.805,E2 -1065.805} C_VEL
LIN {X 0,Y 594.441,Z 524.582,A -85,B 0,C 180,E1 -1066.692,E2 -1066.692} C_VEL
LIN {X 0,Y 594.762,Z 528.792,A -85,B 0,C 180,E1 -1066.765,E2 -1066.765} C_VEL
LIN {X 0,Y 594.695,Z 632.954,A -85,B 0,C 180,E1 -1068.043,E2 -1068.043} C_VEL
LIN {X 0,Y 594.617,Z 645.621,A -85,B 0,C 180,E1 -1068.322,E2 -1068.322} C_VEL
LIN {X 0,Y 594.561,Z 658.367,A -85,B 0,C 180,E1 -1068.746,E2 -1068.746} C_VEL
LIN {X 0,Y 594.532,Z 669.959,A -85,B 0,C 180,E1 -1069.27,E2 -1069.27} C_VEL
LIN {X 0,Y 594.447,Z 680.409,A -85,B 0,C 180,E1 -1069.871,E2 -1069.871} C_VEL
LIN {X 0,Y 594.407,Z 691.188,A -85,B 0,C 180,E1 -1070.644,E2 -1070.644} C_VEL
LIN {X 0,Y 594.384,Z 700.856,A -85,B 0,C 180,E1 -1071.5,E2 -1071.5} C_VEL
LIN {X 0,Y 594.337,Z 710.178,A -85,B 0,C 180,E1 -1072.526,E2 -1072.526} C_VEL
LIN {X 0,Y 594.285,Z 718.061,A -85,B 0,C 180,E1 -1073.613,E2 -1073.613} C_VEL
LIN {X 0,Y 594.289,Z 723.639,A -85,B 0,C 180,E1 -1074.571,E2 -1074.571} C_VEL
LIN {X 0,Y 594.27,Z 728.381,A -85,B 0,C 180,E1 -1075.591,E2 -1075.591} C_VEL
LIN {X 0,Y 594.268,Z 732.019,A -85,B 0,C 180,E1 -1076.61,E2 -1076.61} C_VEL
LIN {X 0,Y 594.225,Z 733.903,A -85,B 0,C 180,E1 -1077.288,E2 -1077.288} C_VEL
LIN {X 0,Y 594.24,Z 735.34,A -85,B 0,C 180,E1 -1077.967,E2 -1077.967} C_VEL
LIN {X 0,Y 594.24,Z 736.963,A -85,B 0,C 180,E1 -1079.322,E2 -1079.322} C_VEL
LIN {X 0,Y 594.236,Z 737.206,A -85,B 0,C 180,E1 -1080,E2 -1080} C_VEL
LIN {X 0,Y 594.24,Z 737.025,A -85,B 0,C 180,E1 -1080.678,E2 -1080.678} C_VEL
LIN {X 0,Y 594.239,Z 735.487,A -85,B 0,C 180,E1 -1082.033,E2 -1082.033} C_VEL
LIN {X 0,Y 594.226,Z 734.11,A -85,B 0,C 180,E1 -1082.712,E2 -1082.712} C_VEL
LIN {X 0,Y 594.289,Z 731.235,A -85,B 0,C 180,E1 -1083.729,E2 -1083.729} C_VEL
LIN {X 0,Y 594.241,Z 727.335,A -85,B 0,C 180,E1 -1084.749,E2 -1084.749} C_VEL
LIN {X 0,Y 594.299,Z 722.307,A -85,B 0,C 180,E1 -1085.769,E2 -1085.769} C_VEL
LIN {X 0,Y 594.317,Z 715.996,A -85,B 0,C 180,E1 -1086.791,E2 -1086.791} C_VEL
LIN {X 0,Y 594.346,Z 708.082,A -85,B 0,C 180,E1 -1087.815,E2 -1087.815} C_VEL
LIN {X 0,Y 594.366,Z 700.014,A -85,B 0,C 180,E1 -1088.671,E2 -1088.671} C_VEL
LIN {X 0,Y 594.416,Z 690.16,A -85,B 0,C 180,E1 -1089.528,E2 -1089.528} C_VEL
LIN {X 0,Y 594.461,Z 679.123,A -85,B 0,C 180,E1 -1090.301,E2 -1090.301} C_VEL
LIN {X 0,Y 594.556,Z 666.67,A -85,B 0,C 180,E1 -1090.983,E2 -1090.983} C_VEL
LIN {X 0,Y 594.582,Z 655.137,A -85,B 0,C 180,E1 -1091.466,E2 -1091.466} C_VEL
LIN {X 0,Y 594.626,Z 642.431,A -85,B 0,C 180,E1 -1091.85,E2 -1091.85} C_VEL
LIN {X 0,Y 594.692,Z 628.935,A -85,B 0,C 180,E1 -1092.109,E2 -1092.109} C_VEL
LIN {X 0,Y 594.646,Z 526.039,A -85,B 0,C 180,E1 -1093.361,E2 -1093.361} C_VEL
LIN {X 0,Y 594.412,Z 524.606,A -85,B 0,C 180,E1 -1093.395,E2 -1093.395} C_VEL
LIN {X 0,Y 594.515,Z 503.653,A -85,B 0,C 180,E1 -1096.129,E2 -1096.129} C_VEL
LIN {X 0,Y 594.621,Z 482.843,A -85,B 0,C 180,E1 -1098.881,E2 -1098.881} C_VEL
LIN {X 0,Y 594.766,Z 462.078,A -85,B 0,C 180,E1 -1101.67,E2 -1101.67} C_VEL
LIN {X 0,Y 594.777,Z 450.008,A -85,B 0,C 180,E1 -1103.318,E2 -1103.318} C_VEL
LIN {X 0,Y 594.407,Z 448.069,A -85,B 0,C 180,E1 -1103.611,E2 -1103.611} C_VEL
LIN {X 0,Y 594.387,Z 448.069,A -85,B 0,C 180,E1 -1106.699,E2 -1106.699} C_VEL
LIN {X 0,Y 594.387,Z 448.066,A -85,B 0,C 180,E1 -1108.998,E2 -1108.998} C_VEL
LIN {X 0,Y 594.382,Z 448.069,A -85,B 0,C 180,E1 -1111.643,E2 -1111.643} C_VEL
LIN {X 0,Y 594.399,Z 448.066,A -85,B 0,C 180,E1 -1114.579,E2 -1114.579} C_VEL
LIN {X 0,Y 594.387,Z 448.065,A -85,B 0,C 180,E1 -1117.087,E2 -1117.087} C_VEL
LIN {X 0,Y 594.364,Z 448.075,A -85,B 0,C 180,E1 -1119.772,E2 -1119.772} C_VEL
LIN {X 0,Y 594.37,Z 448.07,A -85,B 0,C 180,E1 -1122.375,E2 -1122.375} C_VEL
LIN {X 0,Y 594.36,Z 448.07,A -85,B 0,C 180,E1 -1125.192,E2 -1125.192} C_VEL
LIN {X 0,Y 594.373,Z 448.075,A -85,B 0,C 180,E1 -1127.624,E2 -1127.624} C_VEL
LIN {X 0,Y 594.375,Z 448.068,A -85,B 0,C 180,E1 -1130.319,E2 -1130.319} C_VEL
LIN {X 0,Y 594.387,Z 448.066,A -85,B 0,C 180,E1 -1132.913,E2 -1132.913} C_VEL
LIN {X 0,Y 594.386,Z 448.07,A -85,B 0,C 180,E1 -1135.861,E2 -1135.861} C_VEL
LIN {X 0,Y 594.375,Z 448.067,A -85,B 0,C 180,E1 -1138.649,E2 -1138.649} C_VEL
LIN {X 0,Y 594.388,Z 448.07,A -85,B 0,C 180,E1 -1141.042,E2 -1141.042} C_VEL
LIN {X 0,Y 594.384,Z 448.068,A -85,B 0,C 180,E1 -1143.978,E2 -1143.978} C_VEL
LIN {X 0,Y 594.45,Z 448.174,A -85,B 0,C 180,E1 -1145.814,E2 -1145.814} C_VEL
LIN {X 0,Y 595.027,Z 450.9,A -85,B 0,C 180,E1 -1146.137,E2 -1146.137} C_VEL
LIN {X 0,Y 594.914,Z 474.388,A -85,B 0,C 180,E1 -1148.674,E2 -1148.674} C_VEL
LIN {X 0,Y 594.717,Z 500.031,A -85,B 0,C 180,E1 -1151.393,E2 -1151.393} C_VEL
LIN {X 0,Y 594.625,Z 523.326,A -85,B 0,C 180,E1 -1153.829,E2 -1153.829} C_VEL
LIN {X 0,Y 595.02,Z 526.764,A -85,B 0,C 180,E1 -1153.884,E2 -1153.884} C_VEL
LIN {X 0,Y 594.858,Z 662.845,A -85,B 0,C 180,E1 -1155.568,E2 -1155.568} C_VEL
LIN {X 0,Y 594.806,Z 677.226,A -85,B 0,C 180,E1 -1155.891,E2 -1155.891} C_VEL
LIN {X 0,Y 594.735,Z 690.693,A -85,B 0,C 180,E1 -1156.329,E2 -1156.329} C_VEL
LIN {X 0,Y 594.654,Z 704.619,A -85,B 0,C 180,E1 -1156.936,E2 -1156.936} C_VEL
LIN {X 0,Y 594.582,Z 717.082,A -85,B 0,C 180,E1 -1157.628,E2 -1157.628} C_VEL
LIN {X 0,Y 594.515,Z 728.463,A -85,B 0,C 180,E1 -1158.406,E2 -1158.406} C_VEL
LIN {X 0,Y 594.475,Z 738.923,A -85,B 0,C 180,E1 -1159.268,E2 -1159.268} C_VEL
LIN {X 0,Y 594.391,Z 749.326,A -85,B 0,C 180,E1 -1160.299,E2 -1160.299} C_VEL
LIN {X 0,Y 594.355,Z 757.907,A -85,B 0,C 180,E1 -1161.328,E2 -1161.328} C_VEL
LIN {X 0,Y 594.314,Z 766.109,A -85,B 0,C 180,E1 -1162.525,E2 -1162.525} C_VEL
LIN {X 0,Y 594.27,Z 772.233,A -85,B 0,C 180,E1 -1163.619,E2 -1163.619} C_VEL
LIN {X 0,Y 594.247,Z 777.958,A -85,B 0,C 180,E1 -1164.91,E2 -1164.91} C_VEL
LIN {X 0,Y 594.259,Z 781.439,A -85,B 0,C 180,E1 -1165.93,E2 -1165.93} C_VEL
LIN {X 0,Y 594.224,Z 784.829,A -85,B 0,C 180,E1 -1167.288,E2 -1167.288} C_VEL
LIN {X 0,Y 594.241,Z 786.83,A -85,B 0,C 180,E1 -1168.644,E2 -1168.644} C_VEL
LIN {X 0,Y 594.234,Z 787.5,A -85,B 0,C 180,E1 -1169.999,E2 -1169.999} C_VEL
LIN {X 0,Y 594.241,Z 786.832,A -85,B 0,C 180,E1 -1171.354,E2 -1171.354} C_VEL
LIN {X 0,Y 594.224,Z 784.834,A -85,B 0,C 180,E1 -1172.711,E2 -1172.711} C_VEL
LIN {X 0,Y 594.259,Z 781.445,A -85,B 0,C 180,E1 -1174.068,E2 -1174.068} C_VEL
LIN {X 0,Y 594.274,Z 776.572,A -85,B 0,C 180,E1 -1175.428,E2 -1175.428} C_VEL
LIN {X 0,Y 594.299,Z 771.036,A -85,B 0,C 180,E1 -1176.606,E2 -1176.606} C_VEL
LIN {X 0,Y 594.315,Z 763.926,A -85,B 0,C 180,E1 -1177.815,E2 -1177.815} C_VEL
LIN {X 0,Y 594.369,Z 755.206,A -85,B 0,C 180,E1 -1179.013,E2 -1179.013} C_VEL
LIN {X 0,Y 594.399,Z 746.091,A -85,B 0,C 180,E1 -1180.043,E2 -1180.043} C_VEL
LIN {X 0,Y 594.477,Z 735.71,A -85,B 0,C 180,E1 -1181.017,E2 -1181.017} C_VEL
LIN {X 0,Y 594.573,Z 723.72,A -85,B 0,C 180,E1 -1181.937,E2 -1181.937} C_VEL
LIN {X 0,Y 594.616,Z 711.23,A -85,B 0,C 180,E1 -1182.716,E2 -1182.716} C_VEL
LIN {X 0,Y 594.696,Z 699.152,A -85,B 0,C 180,E1 -1183.322,E2 -1183.322} C_VEL
LIN {X 0,Y 594.784,Z 685.231,A -85,B 0,C 180,E1 -1183.865,E2 -1183.865} C_VEL
LIN {X 0,Y 594.799,Z 670.737,A -85,B 0,C 180,E1 -1184.273,E2 -1184.273} C_VEL
LIN {X 0,Y 594.875,Z 655.68,A -85,B 0,C 180,E1 -1184.539,E2 -1184.539} C_VEL
LIN {X 0,Y 594.872,Z 524.9,A -85,B 0,C 180,E1 -1186.143,E2 -1186.143} C_VEL
LIN {X 0,Y 594.625,Z 523.343,A -85,B 0,C 180,E1 -1186.169,E2 -1186.169} C_VEL
LIN {X 0,Y 594.765,Z 495.958,A -85,B 0,C 180,E1 -1189.036,E2 -1189.036} C_VEL
LIN {X 0,Y 594.966,Z 469.553,A -85,B 0,C 180,E1 -1191.843,E2 -1191.843} C_VEL
LIN {X 0,Y 595.025,Z 450.917,A -85,B 0,C 180,E1 -1193.861,E2 -1193.861} C_VEL
LIN {X 0,Y 594.422,Z 448.068,A -85,B 0,C 180,E1 -1194.208,E2 -1194.208} C_VEL
LIN {X 0,Y 594.388,Z 448.075,A -85,B 0,C 180,E1 -1196.698,E2 -1196.698} C_VEL
LIN {X 0,Y 594.38,Z 448.071,A -85,B 0,C 180,E1 -1198.997,E2 -1198.997} C_VEL
LIN {X 0,Y 594.39,Z 448.064,A -85,B 0,C 180,E1 -1201.644,E2 -1201.644} C_VEL
LIN {X 0,Y 594.395,Z 448.072,A -85,B 0,C 180,E1 -1204.577,E2 -1204.577} C_VEL
LIN {X 0,Y 594.385,Z 448.069,A -85,B 0,C 180,E1 -1207.085,E2 -1207.085} C_VEL
LIN {X 0,Y 594.374,Z 448.066,A -85,B 0,C 180,E1 -1209.774,E2 -1209.774} C_VEL
LIN {X 0,Y 594.384,Z 448.07,A -85,B 0,C 180,E1 -1212.372,E2 -1212.372} C_VEL
LIN {X 0,Y 594.355,Z 448.071,A -85,B 0,C 180,E1 -1215.19,E2 -1215.19} C_VEL
LIN {X 0,Y 594.363,Z 448.067,A -85,B 0,C 180,E1 -1217.624,E2 -1217.624} C_VEL
LIN {X 0,Y 594.39,Z 448.068,A -85,B 0,C 180,E1 -1220.321,E2 -1220.321} C_VEL
LIN {X 0,Y 594.381,Z 448.07,A -85,B 0,C 180,E1 -1222.913,E2 -1222.913} C_VEL
LIN {X 0,Y 594.382,Z 448.065,A -85,B 0,C 180,E1 -1225.859,E2 -1225.859} C_VEL
LIN {X 0,Y 594.385,Z 448.075,A -85,B 0,C 180,E1 -1228.651,E2 -1228.651} C_VEL
LIN {X 0,Y 594.382,Z 448.069,A -85,B 0,C 180,E1 -1231.04,E2 -1231.04} C_VEL
LIN {X 0,Y 594.388,Z 448.065,A -85,B 0,C 180,E1 -1233.974,E2 -1233.974} C_VEL
LIN {X 0,Y 594.386,Z 448.069,A -85,B 0,C 180,E1 -1236.296,E2 -1236.296} C_VEL
LIN {X 0,Y 594.401,Z 448.064,A -85,B 0,C 180,E1 -1239.224,E2 -1239.224} C_VEL
LIN {X 0,Y 594.377,Z 448.068,A -85,B 0,C 180,E1 -1242.096,E2 -1242.096} C_VEL
LIN {X 0,Y 594.365,Z 448.071,A -85,B 0,C 180,E1 -1244.219,E2 -1244.219} C_VEL
LIN {X 0,Y 594.368,Z 448.07,A -85,B 0,C 180,E1 -1247.017,E2 -1247.017} C_VEL
LIN {X 0,Y 594.389,Z 448.064,A -85,B 0,C 180,E1 -1249.784,E2 -1249.784} C_VEL
LIN {X 0,Y 594.41,Z 448.071,A -85,B 0,C 180,E1 -1252.527,E2 -1252.527} C_VEL
LIN {X 0,Y 594.398,Z 448.064,A -85,B 0,C 180,E1 -1255.253,E2 -1255.253} C_VEL
LIN {X 0,Y 594.388,Z 448.066,A -85,B 0,C 180,E1 -1257.967,E2 -1257.967} C_VEL
LIN {X 0,Y 594.421,Z 448.069,A -85,B 0,C 180,E1 -1260.678,E2 -1260.678} C_VEL
LIN {X 0,Y 594.378,Z 448.065,A -85,B 0,C 180,E1 -1263.389,E2 -1263.389} C_VEL
LIN {X 0,Y 594.362,Z 448.071,A -85,B 0,C 180,E1 -1266.109,E2 -1266.109} C_VEL
LIN {X 0,Y 594.394,Z 448.069,A -85,B 0,C 180,E1 -1268.842,E2 -1268.842} C_VEL
LIN {X 0,Y 594.385,Z 448.065,A -85,B 0,C 180,E1 -1271.596,E2 -1271.596} C_VEL
LIN {X 0,Y 594.38,Z 448.072,A -85,B 0,C 180,E1 -1274.377,E2 -1274.377} C_VEL
LIN {X 0,Y 594.356,Z 448.069,A -85,B 0,C 180,E1 -1275.341,E2 -1275.341} C_VEL
LIN {X 0,Y 593.686,Z 448.154,A -85,B 0,C 180,E1 -1275.906,E2 -1275.906} C_VEL
LIN {X 0,Y 590.832,Z 448.512,A -85,B 0,C 180,E1 -1276.825,E2 -1276.825} C_VEL
LIN {X 0,Y 588.426,Z 448.811,A -85,B 0,C 180,E1 -1277.563,E2 -1277.563} C_VEL
LIN {X 0,Y 587.4,Z 448.938,A -85,B 0,C 180,E1 -1278.134,E2 -1278.134} C_VEL
LIN {X 0,Y 587.319,Z 448.947,A -85,B 0,C 180,E1 -1278.327,E2 -1278.327} C_VEL
LIN {X 0,Y 587.348,Z 448.944,A -85,B 0,C 180,E1 -1281.045,E2 -1281.045} C_VEL
LIN {X 0,Y 587.33,Z 448.946,A -85,B 0,C 180,E1 -1284.007,E2 -1284.007} C_VEL
LIN {X 0,Y 587.357,Z 448.946,A -85,B 0,C 180,E1 -1286.278,E2 -1286.278} C_VEL
LIN {X 0,Y 587.347,Z 448.943,A -85,B 0,C 180,E1 -1289.136,E2 -1289.136} C_VEL
LIN {X 0,Y 587.35,Z 448.942,A -85,B 0,C 180,E1 -1291.839,E2 -1291.839} C_VEL
LIN {X 0,Y 587.352,Z 448.948,A -85,B 0,C 180,E1 -1294.351,E2 -1294.351} C_VEL
LIN {X 0,Y 587.346,Z 448.947,A -85,B 0,C 180,E1 -1296.747,E2 -1296.747} C_VEL
LIN {X 0,Y 587.343,Z 448.942,A -85,B 0,C 180,E1 -1299.36,E2 -1299.36} C_VEL
LIN {X 0,Y 587.327,Z 448.948,A -85,B 0,C 180,E1 -1302.109,E2 -1302.109} C_VEL
LIN {X 0,Y 587.31,Z 448.948,A -85,B 0,C 180,E1 -1305.09,E2 -1305.09} C_VEL
LIN {X 0,Y 587.347,Z 448.944,A -85,B 0,C 180,E1 -1307.929,E2 -1307.929} C_VEL
LIN {X 0,Y 587.332,Z 448.945,A -85,B 0,C 180,E1 -1311.059,E2 -1311.059} C_VEL
LIN {X 0,Y 587.351,Z 448.941,A -85,B 0,C 180,E1 -1313.293,E2 -1313.293} C_VEL
LIN {X 0,Y 587.365,Z 448.941,A -85,B 0,C 180,E1 -1315.782,E2 -1315.782} C_VEL
LIN {X 0,Y 587.353,Z 448.948,A -85,B 0,C 180,E1 -1318.233,E2 -1318.233} C_VEL
LIN {X 0,Y 587.349,Z 448.946,A -85,B 0,C 180,E1 -1320.867,E2 -1320.867} C_VEL
LIN {X 0,Y 587.361,Z 448.943,A -85,B 0,C 180,E1 -1323.819,E2 -1323.819} C_VEL
LIN {X 0,Y 587.339,Z 448.948,A -85,B 0,C 180,E1 -1325.995,E2 -1325.995} C_VEL
LIN {X 0,Y 587.332,Z 449.007,A -85,B 0,C 180,E1 -1327.129,E2 -1327.129} C_VEL
LIN {X 0,Y 587.844,Z 454.002,A -85,B 0,C 180,E1 -1327.878,E2 -1327.878} C_VEL
LIN {X 0,Y 587.677,Z 474.82,A -85,B 0,C 180,E1 -1330.867,E2 -1330.867} C_VEL
LIN {X 0,Y 587.532,Z 494.71,A -85,B 0,C 180,E1 -1333.675,E2 -1333.675} C_VEL
LIN {X 0,Y 587.425,Z 515.225,A -85,B 0,C 180,E1 -1336.532,E2 -1336.532} C_VEL
LIN {X 0,Y 587.866,Z 519.224,A -85,B 0,C 180,E1 -1336.608,E2 -1336.608} C_VEL
LIN {X 0,Y 587.746,Z 623.437,A -85,B 0,C 180,E1 -1337.9,E2 -1337.9} C_VEL
LIN {X 0,Y 587.683,Z 636.707,A -85,B 0,C 180,E1 -1338.205,E2 -1338.205} C_VEL
LIN {X 0,Y 587.608,Z 649.308,A -85,B 0,C 180,E1 -1338.637,E2 -1338.637} C_VEL
LIN {X 0,Y 587.573,Z 660.294,A -85,B 0,C 180,E1 -1339.142,E2 -1339.142} C_VEL
LIN {X 0,Y 587.474,Z 672.054,A -85,B 0,C 180,E1 -1339.838,E2 -1339.838} C_VEL
LIN {X 0,Y 587.393,Z 682.56,A -85,B 0,C 180,E1 -1340.619,E2 -1340.619} C_VEL
LIN {X 0,Y 587.323,Z 691.161,A -85,B 0,C 180,E1 -1341.399,E2 -1341.399} C_VEL
LIN {X 0,Y 587.274,Z 699.086,A -85,B 0,C 180,E1 -1342.264,E2 -1342.264} C_VEL
LIN {X 0,Y 587.235,Z 705.656,A -85,B 0,C 180,E1 -1343.127,E2 -1343.127} C_VEL
LIN {X 0,Y 587.237,Z 712.124,A -85,B 0,C 180,E1 -1344.162,E2 -1344.162} C_VEL
LIN {X 0,Y 587.146,Z 717.262,A -85,B 0,C 180,E1 -1345.195,E2 -1345.195} C_VEL
LIN {X 0,Y 587.212,Z 721.251,A -85,B 0,C 180,E1 -1346.227,E2 -1346.227} C_VEL
LIN {X 0,Y 587.131,Z 724.199,A -85,B 0,C 180,E1 -1347.257,E2 -1347.257} C_VEL
LIN {X 0,Y 587.14,Z 725.629,A -85,B 0,C 180,E1 -1347.943,E2 -1347.943} C_VEL
LIN {X 0,Y 587.14,Z 727.254,A -85,B 0,C 180,E1 -1349.315,E2 -1349.315} C_VEL
LIN {X 0,Y 587.137,Z 727.496,A -85,B 0,C 180,E1 -1350.001,E2 -1350.001} C_VEL
LIN {X 0,Y 587.14,Z 727.314,A -85,B 0,C 180,E1 -1350.687,E2 -1350.687} C_VEL
LIN {X 0,Y 587.14,Z 725.773,A -85,B 0,C 180,E1 -1352.059,E2 -1352.059} C_VEL
LIN {X 0,Y 587.133,Z 724.411,A -85,B 0,C 180,E1 -1352.745,E2 -1352.745} C_VEL
LIN {X 0,Y 587.213,Z 721.533,A -85,B 0,C 180,E1 -1353.775,E2 -1353.775} C_VEL
LIN {X 0,Y 587.147,Z 717.633,A -85,B 0,C 180,E1 -1354.807,E2 -1354.807} C_VEL
LIN {X 0,Y 587.229,Z 712.6,A -85,B 0,C 180,E1 -1355.84,E2 -1355.84} C_VEL
LIN {X 0,Y 587.231,Z 706.278,A -85,B 0,C 180,E1 -1356.874,E2 -1356.874} C_VEL
LIN {X 0,Y 587.288,Z 698.358,A -85,B 0,C 180,E1 -1357.911,E2 -1357.911} C_VEL
LIN {X 0,Y 587.344,Z 688.509,A -85,B 0,C 180,E1 -1358.95,E2 -1358.95} C_VEL
LIN {X 0,Y 587.418,Z 678.185,A -85,B 0,C 180,E1 -1359.817,E2 -1359.817} C_VEL
LIN {X 0,Y 587.527,Z 666.555,A -85,B 0,C 180,E1 -1360.599,E2 -1360.599} C_VEL
LIN {X 0,Y 587.594,Z 655.581,A -85,B 0,C 180,E1 -1361.181,E2 -1361.181} C_VEL
LIN {X 0,Y 587.626,Z 643.038,A -85,B 0,C 180,E1 -1361.686,E2 -1361.686} C_VEL
LIN {X 0,Y 587.711,Z 629.956,A -85,B 0,C 180,E1 -1362.058,E2 -1362.058} C_VEL
LIN {X 0,Y 587.751,Z 617.613,A -85,B 0,C 180,E1 -1362.277,E2 -1362.277} C_VEL
LIN {X 0,Y 587.732,Z 517.447,A -85,B 0,C 180,E1 -1363.507,E2 -1363.507} C_VEL
LIN {X 0,Y 587.406,Z 515.225,A -85,B 0,C 180,E1 -1363.559,E2 -1363.559} C_VEL
LIN {X 0,Y 587.534,Z 495.339,A -85,B 0,C 180,E1 -1366.327,E2 -1366.327} C_VEL
LIN {X 0,Y 587.675,Z 475.457,A -85,B 0,C 180,E1 -1369.132,E2 -1369.132} C_VEL
LIN {X 0,Y 587.851,Z 454.608,A -85,B 0,C 180,E1 -1372.124,E2 -1372.124} C_VEL
LIN {X 0,Y 587.417,Z 449.466,A -85,B 0,C 180,E1 -1372.89,E2 -1372.89} C_VEL
LIN {X 0,Y 587.332,Z 448.951,A -85,B 0,C 180,E1 -1373.025,E2 -1373.025} C_VEL
LIN {X 0,Y 587.341,Z 448.952,A -85,B 0,C 180,E1 -1375.517,E2 -1375.517} C_VEL
LIN {X 0,Y 587.354,Z 448.95,A -85,B 0,C 180,E1 -1377.818,E2 -1377.818} C_VEL
LIN {X 0,Y 587.345,Z 448.943,A -85,B 0,C 180,E1 -1380.511,E2 -1380.511} C_VEL
LIN {X 0,Y 587.341,Z 448.948,A -85,B 0,C 180,E1 -1383.397,E2 -1383.397} C_VEL
LIN {X 0,Y 587.297,Z 448.954,A -85,B 0,C 180,E1 -1385.9,E2 -1385.9} C_VEL
LIN {X 0,Y 587.338,Z 448.943,A -85,B 0,C 180,E1 -1388.479,E2 -1388.479} C_VEL
LIN {X 0,Y 587.342,Z 448.945,A -85,B 0,C 180,E1 -1391.157,E2 -1391.157} C_VEL
LIN {X 0,Y 587.341,Z 448.945,A -85,B 0,C 180,E1 -1394.114,E2 -1394.114} C_VEL
LIN {X 0,Y 587.319,Z 448.946,A -85,B 0,C 180,E1 -1396.994,E2 -1396.994} C_VEL
LIN {X 0,Y 587.319,Z 448.955,A -85,B 0,C 180,E1 -1399.746,E2 -1399.746} C_VEL
LIN {X 0,Y 587.349,Z 448.942,A -85,B 0,C 180,E1 -1402.392,E2 -1402.392} C_VEL
LIN {X 0,Y 587.354,Z 448.941,A -85,B 0,C 180,E1 -1404.946,E2 -1404.946} C_VEL
LIN {X 0,Y 587.344,Z 448.948,A -85,B 0,C 180,E1 -1407.421,E2 -1407.421} C_VEL
LIN {X 0,Y 587.339,Z 448.951,A -85,B 0,C 180,E1 -1409.83,E2 -1409.83} C_VEL
LIN {X 0,Y 587.347,Z 448.943,A -85,B 0,C 180,E1 -1412.309,E2 -1412.309} C_VEL
LIN {X 0,Y 587.341,Z 448.944,A -85,B 0,C 180,E1 -1414.483,E2 -1414.483} C_VEL
LIN {X 0,Y 587.369,Z 449.021,A -85,B 0,C 180,E1 -1416.323,E2 -1416.323} C_VEL
LIN {X 0,Y 587.936,Z 453.647,A -85,B 0,C 180,E1 -1416.99,E2 -1416.99} C_VEL
LIN {X 0,Y 587.735,Z 474.822,A -85,B 0,C 180,E1 -1419.892,E2 -1419.892} C_VEL
LIN {X 0,Y 587.589,Z 494.928,A -85,B 0,C 180,E1 -1422.601,E2 -1422.601} C_VEL
LIN {X 0,Y 587.482,Z 516.376,A -85,B 0,C 180,E1 -1425.45,E2 -1425.45} C_VEL
LIN {X 0,Y 587.42,Z 524.67,A -85,B 0,C 180,E1 -1426.541,E2 -1426.541} C_VEL
LIN {X 0,Y 587.851,Z 528.837,A -85,B 0,C 180,E1 -1426.606,E2 -1426.606} C_VEL
LIN {X 0,Y 587.748,Z 632.94,A -85,B 0,C 180,E1 -1427.899,E2 -1427.899} C_VEL
LIN {X 0,Y 587.663,Z 645.648,A -85,B 0,C 180,E1 -1428.182,E2 -1428.182} C_VEL
LIN {X 0,Y 587.597,Z 659.3,A -85,B 0,C 180,E1 -1428.647,E2 -1428.647} C_VEL
LIN {X 0,Y 587.532,Z 671.567,A -85,B 0,C 180,E1 -1429.228,E2 -1429.228} C_VEL
LIN {X 0,Y 587.46,Z 681.731,A -85,B 0,C 180,E1 -1429.836,E2 -1429.836} C_VEL
LIN {X 0,Y 587.395,Z 692.255,A -85,B 0,C 180,E1 -1430.618,E2 -1430.618} C_VEL
LIN {X 0,Y 587.341,Z 702.571,A -85,B 0,C 180,E1 -1431.571,E2 -1431.571} C_VEL
LIN {X 0,Y 587.26,Z 711.539,A -85,B 0,C 180,E1 -1432.608,E2 -1432.608} C_VEL
LIN {X 0,Y 587.198,Z 718.63,A -85,B 0,C 180,E1 -1433.625,E2 -1433.625} C_VEL
LIN {X 0,Y 587.211,Z 723.636,A -85,B 0,C 180,E1 -1434.506,E2 -1434.506} C_VEL
LIN {X 0,Y 587.188,Z 728.378,A -85,B 0,C 180,E1 -1435.538,E2 -1435.538} C_VEL
LIN {X 0,Y 587.194,Z 732.018,A -85,B 0,C 180,E1 -1436.569,E2 -1436.569} C_VEL
LIN {X 0,Y 587.132,Z 733.899,A -85,B 0,C 180,E1 -1437.256,E2 -1437.256} C_VEL
LIN {X 0,Y 587.139,Z 735.342,A -85,B 0,C 180,E1 -1437.942,E2 -1437.942} C_VEL
LIN {X 0,Y 587.14,Z 736.964,A -85,B 0,C 180,E1 -1439.314,E2 -1439.314} C_VEL
LIN {X 0,Y 587.137,Z 737.206,A -85,B 0,C 180,E1 -1440,E2 -1440} C_VEL
LIN {X 0,Y 587.147,Z 736.443,A -85,B 0,C 180,E1 -1441.372,E2 -1441.372} C_VEL
LIN {X 0,Y 587.138,Z 735.487,A -85,B 0,C 180,E1 -1442.058,E2 -1442.058} C_VEL
LIN {X 0,Y 587.132,Z 734.102,A -85,B 0,C 180,E1 -1442.744,E2 -1442.744} C_VEL
LIN {X 0,Y 587.213,Z 731.227,A -85,B 0,C 180,E1 -1443.774,E2 -1443.774} C_VEL
LIN {X 0,Y 587.146,Z 727.327,A -85,B 0,C 180,E1 -1444.806,E2 -1444.806} C_VEL
LIN {X 0,Y 587.229,Z 722.301,A -85,B 0,C 180,E1 -1445.839,E2 -1445.839} C_VEL
LIN {X 0,Y 587.23,Z 715.991,A -85,B 0,C 180,E1 -1446.874,E2 -1446.874} C_VEL
LIN {X 0,Y 587.288,Z 708.079,A -85,B 0,C 180,E1 -1447.91,E2 -1447.91} C_VEL
LIN {X 0,Y 587.325,Z 700.009,A -85,B 0,C 180,E1 -1448.776,E2 -1448.776} C_VEL
LIN {X 0,Y 587.386,Z 690.141,A -85,B 0,C 180,E1 -1449.643,E2 -1449.643} C_VEL
LIN {X 0,Y 587.478,Z 679.116,A -85,B 0,C 180,E1 -1450.424,E2 -1450.424} C_VEL
LIN {X 0,Y 587.578,Z 666.722,A -85,B 0,C 180,E1 -1451.112,E2 -1451.112} C_VEL
LIN {X 0,Y 587.616,Z 654.05,A -85,B 0,C 180,E1 -1451.64,E2 -1451.64} C_VEL
LIN {X 0,Y 587.718,Z 641.506,A -85,B 0,C 180,E1 -1452.014,E2 -1452.014} C_VEL
LIN {X 0,Y 587.773,Z 628.897,A -85,B 0,C 180,E1 -1452.253,E2 -1452.253} C_VEL
LIN {X 0,Y 587.746,Z 526.776,A -85,B 0,C 180,E1 -1453.511,E2 -1453.511} C_VEL
LIN {X 0,Y 587.418,Z 524.602,A -85,B 0,C 180,E1 -1453.558,E2 -1453.558} C_VEL
LIN {X 0,Y 587.551,Z 503.648,A -85,B 0,C 180,E1 -1456.326,E2 -1456.326} C_VEL
LIN {X 0,Y 587.694,Z 481.538,A -85,B 0,C 180,E1 -1459.288,E2 -1459.288} C_VEL
LIN {X 0,Y 587.92,Z 459.392,A -85,B 0,C 180,E1 -1462.305,E2 -1462.305} C_VEL
LIN {X 0,Y 587.835,Z 451.344,A -85,B 0,C 180,E1 -1463.424,E2 -1463.424} C_VEL
LIN {X 0,Y 587.381,Z 448.946,A -85,B 0,C 180,E1 -1463.794,E2 -1463.794} C_VEL
LIN {X 0,Y 587.345,Z 448.953,A -85,B 0,C 180,E1 -1466.278,E2 -1466.278} C_VEL
LIN {X 0,Y 587.355,Z 448.942,A -85,B 0,C 180,E1 -1469.133,E2 -1469.133} C_VEL
LIN {X 0,Y 587.349,Z 448.948,A -85,B 0,C 180,E1 -1471.836,E2 -1471.836} C_VEL
LIN {X 0,Y 587.359,Z 448.947,A -85,B 0,C 180,E1 -1474.348,E2 -1474.348} C_VEL
LIN {X 0,Y 587.357,Z 448.942,A -85,B 0,C 180,E1 -1476.746,E2 -1476.746} C_VEL
LIN {X 0,Y 587.338,Z 448.945,A -85,B 0,C 180,E1 -1479.36,E2 -1479.36} C_VEL
LIN {X 0,Y 587.34,Z 448.95,A -85,B 0,C 180,E1 -1482.107,E2 -1482.107} C_VEL
LIN {X 0,Y 587.309,Z 448.948,A -85,B 0,C 180,E1 -1485.087,E2 -1485.087} C_VEL
LIN {X 0,Y 587.343,Z 448.95,A -85,B 0,C 180,E1 -1487.926,E2 -1487.926} C_VEL
LIN {X 0,Y 587.327,Z 448.946,A -85,B 0,C 180,E1 -1491.059,E2 -1491.059} C_VEL
LIN {X 0,Y 587.352,Z 448.946,A -85,B 0,C 180,E1 -1493.292,E2 -1493.292} C_VEL
LIN {X 0,Y 587.366,Z 448.946,A -85,B 0,C 180,E1 -1495.78,E2 -1495.78} C_VEL
LIN {X 0,Y 587.346,Z 448.943,A -85,B 0,C 180,E1 -1498.231,E2 -1498.231} C_VEL
LIN {X 0,Y 587.354,Z 448.944,A -85,B 0,C 180,E1 -1500.866,E2 -1500.866} C_VEL
LIN {X 0,Y 587.361,Z 448.945,A -85,B 0,C 180,E1 -1503.819,E2 -1503.819} C_VEL
LIN {X 0,Y 587.384,Z 449.034,A -85,B 0,C 180,E1 -1505.6,E2 -1505.6} C_VEL
LIN {X 0,Y 588.199,Z 452.594,A -85,B 0,C 180,E1 -1506.03,E2 -1506.03} C_VEL
LIN {X 0,Y 588.069,Z 474.454,A -85,B 0,C 180,E1 -1508.42,E2 -1508.42} C_VEL
LIN {X 0,Y 587.818,Z 501.725,A -85,B 0,C 180,E1 -1511.347,E2 -1511.347} C_VEL
LIN {X 0,Y 587.681,Z 523.326,A -85,B 0,C 180,E1 -1513.633,E2 -1513.633} C_VEL
LIN {X 0,Y 588.214,Z 528.553,A -85,B 0,C 180,E1 -1513.715,E2 -1513.715} C_VEL
LIN {X 0,Y 587.989,Z 662.845,A -85,B 0,C 180,E1 -1515.396,E2 -1515.396} C_VEL
LIN {X 0,Y 587.915,Z 677.415,A -85,B 0,C 180,E1 -1515.727,E2 -1515.727} C_VEL
LIN {X 0,Y 587.824,Z 691.816,A -85,B 0,C 180,E1 -1516.209,E2 -1516.209} C_VEL
LIN {X 0,Y 587.731,Z 704.621,A -85,B 0,C 180,E1 -1516.779,E2 -1516.779} C_VEL
LIN {X 0,Y 587.605,Z 717.083,A -85,B 0,C 180,E1 -1517.479,E2 -1517.479} C_VEL
LIN {X 0,Y 587.514,Z 728.465,A -85,B 0,C 180,E1 -1518.266,E2 -1518.266} C_VEL
LIN {X 0,Y 587.467,Z 738.924,A -85,B 0,C 180,E1 -1519.139,E2 -1519.139} C_VEL
LIN {X 0,Y 587.353,Z 749.326,A -85,B 0,C 180,E1 -1520.182,E2 -1520.182} C_VEL
LIN {X 0,Y 587.311,Z 757.907,A -85,B 0,C 180,E1 -1521.223,E2 -1521.223} C_VEL
LIN {X 0,Y 587.25,Z 766.11,A -85,B 0,C 180,E1 -1522.435,E2 -1522.435} C_VEL
LIN {X 0,Y 587.179,Z 772.681,A -85,B 0,C 180,E1 -1523.635,E2 -1523.635} C_VEL
LIN {X 0,Y 587.16,Z 777.958,A -85,B 0,C 180,E1 -1524.849,E2 -1524.849} C_VEL
LIN {X 0,Y 587.179,Z 781.439,A -85,B 0,C 180,E1 -1525.881,E2 -1525.881} C_VEL
LIN {X 0,Y 587.13,Z 784.83,A -85,B 0,C 180,E1 -1527.255,E2 -1527.255} C_VEL
LIN {X 0,Y 587.141,Z 786.831,A -85,B 0,C 180,E1 -1528.627,E2 -1528.627} C_VEL
LIN {X 0,Y 587.135,Z 787.5,A -85,B 0,C 180,E1 -1529.999,E2 -1529.999} C_VEL
LIN {X 0,Y 587.141,Z 786.833,A -85,B 0,C 180,E1 -1531.371,E2 -1531.371} C_VEL
LIN {X 0,Y 587.13,Z 784.834,A -85,B 0,C 180,E1 -1532.743,E2 -1532.743} C_VEL
LIN {X 0,Y 587.179,Z 781.446,A -85,B 0,C 180,E1 -1534.117,E2 -1534.117} C_VEL
LIN {X 0,Y 587.199,Z 776.572,A -85,B 0,C 180,E1 -1535.494,E2 -1535.494} C_VEL
LIN {X 0,Y 587.208,Z 770.057,A -85,B 0,C 180,E1 -1536.873,E2 -1536.873} C_VEL
LIN {X 0,Y 587.268,Z 762.805,A -85,B 0,C 180,E1 -1538.082,E2 -1538.082} C_VEL
LIN {X 0,Y 587.33,Z 753.831,A -85,B 0,C 180,E1 -1539.295,E2 -1539.295} C_VEL
LIN {X 0,Y 587.371,Z 744.401,A -85,B 0,C 180,E1 -1540.338,E2 -1540.338} C_VEL
LIN {X 0,Y 587.474,Z 734.035,A -85,B 0,C 180,E1 -1541.29,E2 -1541.29} C_VEL
LIN {X 0,Y 587.578,Z 722.444,A -85,B 0,C 180,E1 -1542.169,E2 -1542.169} C_VEL
LIN {X 0,Y 587.67,Z 709.666,A -85,B 0,C 180,E1 -1542.957,E2 -1542.957} C_VEL
LIN {X 0,Y 587.813,Z 697.184,A -85,B 0,C 180,E1 -1543.569,E2 -1543.569} C_VEL
LIN {X 0,Y 587.9,Z 683.76,A -85,B 0,C 180,E1 -1544.08,E2 -1544.08} C_VEL
LIN {X 0,Y 587.96,Z 669.346,A -85,B 0,C 180,E1 -1544.476,E2 -1544.476} C_VEL
LIN {X 0,Y 588.009,Z 655.68,A -85,B 0,C 180,E1 -1544.712,E2 -1544.712} C_VEL
LIN {X 0,Y 588.12,Z 526.143,A -85,B 0,C 180,E1 -1546.318,E2 -1546.318} C_VEL
LIN {X 0,Y 587.685,Z 523.343,A -85,B 0,C 180,E1 -1546.365,E2 -1546.365} C_VEL
LIN {X 0,Y 587.87,Z 495.627,A -85,B 0,C 180,E1 -1549.303,E2 -1549.303} C_VEL
LIN {X 0,Y 588.114,Z 469.553,A -85,B 0,C 180,E1 -1552.111,E2 -1552.111} C_VEL
LIN {X 0,Y 588.196,Z 452.612,A -85,B 0,C 180,E1 -1553.968,E2 -1553.968} C_VEL
LIN {X 0,Y 587.356,Z 448.95,A -85,B 0,C 180,E1 -1554.42,E2 -1554.42} C_VEL
LIN {X 0,Y 587.33,Z 448.95,A -85,B 0,C 180,E1 -1557.045,E2 -1557.045} C_VEL
LIN {X 0,Y 587.348,Z 448.943,A -85,B 0,C 180,E1 -1559.378,E2 -1559.378} C_VEL
LIN {X 0,Y 587.354,Z 448.941,A -85,B 0,C 180,E1 -1561.837,E2 -1561.837} C_VEL
LIN {X 0,Y 587.353,Z 448.945,A -85,B 0,C 180,E1 -1564.348,E2 -1564.348} C_VEL
LIN {X 0,Y 587.349,Z 448.952,A -85,B 0,C 180,E1 -1566.745,E2 -1566.745} C_VEL
LIN {X 0,Y 587.343,Z 448.943,A -85,B 0,C 180,E1 -1569.358,E2 -1569.358} C_VEL
LIN {X 0,Y 587.36,Z 448.942,A -85,B 0,C 180,E1 -1572.11,E2 -1572.11} C_VEL
LIN {X 0,Y 587.308,Z 448.95,A -85,B 0,C 180,E1 -1575.088,E2 -1575.088} C_VEL
LIN {X 0,Y 587.344,Z 448.942,A -85,B 0,C 180,E1 -1577.927,E2 -1577.927} C_VEL
LIN {X 0,Y 587.33,Z 448.947,A -85,B 0,C 180,E1 -1581.057,E2 -1581.057} C_VEL
LIN {X 0,Y 587.346,Z 448.941,A -85,B 0,C 180,E1 -1583.291,E2 -1583.291} C_VEL
LIN {X 0,Y 587.365,Z 448.939,A -85,B 0,C 180,E1 -1585.78,E2 -1585.78} C_VEL
LIN {X 0,Y 587.347,Z 448.945,A -85,B 0,C 180,E1 -1588.231,E2 -1588.231} C_VEL
LIN {X 0,Y 587.347,Z 448.948,A -85,B 0,C 180,E1 -1590.864,E2 -1590.864} C_VEL
LIN {X 0,Y 587.355,Z 448.941,A -85,B 0,C 180,E1 -1593.817,E2 -1593.817} C_VEL
LIN {X 0,Y 587.316,Z 448.951,A -85,B 0,C 180,E1 -1596.741,E2 -1596.741} C_VEL
LIN {X 0,Y 587.327,Z 448.943,A -85,B 0,C 180,E1 -1599.695,E2 -1599.695} C_VEL
LIN {X 0,Y 587.353,Z 448.951,A -85,B 0,C 180,E1 -1602.594,E2 -1602.594} C_VEL
LIN {X 0,Y 587.354,Z 448.941,A -85,B 0,C 180,E1 -1605.739,E2 -1605.739} C_VEL
LIN {X 0,Y 587.351,Z 448.947,A -85,B 0,C 180,E1 -1608.858,E2 -1608.858} C_VEL
LIN {X 0,Y 587.363,Z 448.94,A -85,B 0,C 180,E1 -1611.745,E2 -1611.745} C_VEL
LIN {X 0,Y 587.355,Z 448.949,A -85,B 0,C 180,E1 -1614.507,E2 -1614.507} C_VEL
LIN {X 0,Y 587.375,Z 448.939,A -85,B 0,C 180,E1 -1617.257,E2 -1617.257} C_VEL
LIN {X 0,Y 587.373,Z 448.94,A -85,B 0,C 180,E1 -1620,E2 -1620} C_VEL
LIN {X 0,Y 587.376,Z 448.944,A -85,B 0,C 180,E1 -1622.743,E2 -1622.743} C_VEL
LIN {X 0,Y 587.349,Z 448.941,A -85,B 0,C 180,E1 -1625.493,E2 -1625.493} C_VEL
LIN {X 0,Y 587.363,Z 448.944,A -85,B 0,C 180,E1 -1628.255,E2 -1628.255} C_VEL
LIN {X 0,Y 587.351,Z 448.943,A -85,B 0,C 180,E1 -1631.142,E2 -1631.142} C_VEL
LIN {X 0,Y 587.354,Z 448.945,A -85,B 0,C 180,E1 -1634.261,E2 -1634.261} C_VEL
LIN {X 0,Y 587.35,Z 448.941,A -85,B 0,C 180,E1 -1637.406,E2 -1637.406} C_VEL
LIN {X 0,Y 587.319,Z 448.947,A -85,B 0,C 180,E1 -1638.327,E2 -1638.327} C_VEL
LIN {X 0,Y 586.667,Z 449.031,A -85,B 0,C 180,E1 -1638.899,E2 -1638.899} C_VEL
LIN {X 0,Y 583.836,Z 449.382,A -85,B 0,C 180,E1 -1639.827,E2 -1639.827} C_VEL
LIN {X 0,Y 581.425,Z 449.689,A -85,B 0,C 180,E1 -1640.574,E2 -1640.574} C_VEL
LIN {X 0,Y 580.372,Z 449.812,A -85,B 0,C 180,E1 -1641.15,E2 -1641.15} C_VEL
LIN {X 0,Y 580.278,Z 449.822,A -85,B 0,C 180,E1 -1641.345,E2 -1641.345} C_VEL
LIN {X 0,Y 580.293,Z 449.827,A -85,B 0,C 180,E1 -1644.317,E2 -1644.317} C_VEL
LIN {X 0,Y 580.3,Z 449.828,A -85,B 0,C 180,E1 -1646.622,E2 -1646.622} C_VEL
LIN {X 0,Y 580.301,Z 449.819,A -85,B 0,C 180,E1 -1649.312,E2 -1649.312} C_VEL
LIN {X 0,Y 580.297,Z 449.825,A -85,B 0,C 180,E1 -1652.201,E2 -1652.201} C_VEL
LIN {X 0,Y 580.296,Z 449.827,A -85,B 0,C 180,E1 -1654.696,E2 -1654.696} C_VEL
LIN {X 0,Y 580.293,Z 449.82,A -85,B 0,C 180,E1 -1657.269,E2 -1657.269} C_VEL
LIN {X 0,Y 580.301,Z 449.826,A -85,B 0,C 180,E1 -1660.274,E2 -1660.274} C_VEL
LIN {X 0,Y 580.272,Z 449.829,A -85,B 0,C 180,E1 -1662.707,E2 -1662.707} C_VEL
LIN {X 0,Y 580.268,Z 449.824,A -85,B 0,C 180,E1 -1665.61,E2 -1665.61} C_VEL
LIN {X 0,Y 580.31,Z 449.825,A -85,B 0,C 180,E1 -1668.236,E2 -1668.236} C_VEL
LIN {X 0,Y 580.287,Z 449.824,A -85,B 0,C 180,E1 -1670.967,E2 -1670.967} C_VEL
LIN {X 0,Y 580.293,Z 449.82,A -85,B 0,C 180,E1 -1673.6,E2 -1673.6} C_VEL
LIN {X 0,Y 580.318,Z 449.823,A -85,B 0,C 180,E1 -1676.147,E2 -1676.147} C_VEL
LIN {X 0,Y 580.29,Z 449.829,A -85,B 0,C 180,E1 -1678.617,E2 -1678.617} C_VEL
LIN {X 0,Y 580.292,Z 449.823,A -85,B 0,C 180,E1 -1681.025,E2 -1681.025} C_VEL
LIN {X 0,Y 580.327,Z 449.818,A -85,B 0,C 180,E1 -1683.66,E2 -1683.66} C_VEL
LIN {X 0,Y 580.28,Z 449.832,A -85,B 0,C 180,E1 -1686.443,E2 -1686.443} C_VEL
LIN {X 0,Y 580.314,Z 450.026,A -85,B 0,C 180,E1 -1686.987,E2 -1686.987} C_VEL
LIN {X 0,Y 580.932,Z 454.006,A -85,B 0,C 180,E1 -1687.601,E2 -1687.601} C_VEL
LIN {X 0,Y 580.755,Z 474.078,A -85,B 0,C 180,E1 -1690.522,E2 -1690.522} C_VEL
LIN {X 0,Y 580.539,Z 494.715,A -85,B 0,C 180,E1 -1693.473,E2 -1693.473} C_VEL
LIN {X 0,Y 580.396,Z 515.07,A -85,B 0,C 180,E1 -1696.343,E2 -1696.343} C_VEL
LIN {X 0,Y 580.425,Z 515.696,A -85,B 0,C 180,E1 -1696.388,E2 -1696.388} C_VEL
LIN {X 0,Y 580.959,Z 521.058,A -85,B 0,C 180,E1 -1696.468,E2 -1696.468} C_VEL
LIN {X 0,Y 580.821,Z 623.465,A -85,B 0,C 180,E1 -1697.754,E2 -1697.754} C_VEL
LIN {X 0,Y 580.757,Z 635.965,A -85,B 0,C 180,E1 -1698.041,E2 -1698.041} C_VEL
LIN {X 0,Y 580.673,Z 648.877,A -85,B 0,C 180,E1 -1698.482,E2 -1698.482} C_VEL
LIN {X 0,Y 580.587,Z 660.307,A -85,B 0,C 180,E1 -1699.01,E2 -1699.01} C_VEL
LIN {X 0,Y 580.454,Z 672.06,A -85,B 0,C 180,E1 -1699.713,E2 -1699.713} C_VEL
LIN {X 0,Y 580.344,Z 682.568,A -85,B 0,C 180,E1 -1700.504,E2 -1700.504} C_VEL
LIN {X 0,Y 580.272,Z 691.167,A -85,B 0,C 180,E1 -1701.293,E2 -1701.293} C_VEL
LIN {X 0,Y 580.221,Z 699.09,A -85,B 0,C 180,E1 -1702.169,E2 -1702.169} C_VEL
LIN {X 0,Y 580.167,Z 706.788,A -85,B 0,C 180,E1 -1703.21,E2 -1703.21} C_VEL
LIN {X 0,Y 580.139,Z 713.952,A -85,B 0,C 180,E1 -1704.439,E2 -1704.439} C_VEL
LIN {X 0,Y 580.108,Z 718.692,A -85,B 0,C 180,E1 -1705.484,E2 -1705.484} C_VEL
LIN {X 0,Y 580.123,Z 722.324,A -85,B 0,C 180,E1 -1706.528,E2 -1706.528} C_VEL
LIN {X 0,Y 580.043,Z 724.201,A -85,B 0,C 180,E1 -1707.223,E2 -1707.223} C_VEL
LIN {X 0,Y 580.039,Z 725.629,A -85,B 0,C 180,E1 -1707.918,E2 -1707.918} C_VEL
LIN {X 0,Y 580.04,Z 727.255,A -85,B 0,C 180,E1 -1709.307,E2 -1709.307} C_VEL
LIN {X 0,Y 580.038,Z 727.496,A -85,B 0,C 180,E1 -1710.001,E2 -1710.001} C_VEL
LIN {X 0,Y 580.04,Z 727.314,A -85,B 0,C 180,E1 -1710.695,E2 -1710.695} C_VEL
LIN {X 0,Y 580.04,Z 725.771,A -85,B 0,C 180,E1 -1712.084,E2 -1712.084} C_VEL
LIN {X 0,Y 580.044,Z 724.409,A -85,B 0,C 180,E1 -1712.779,E2 -1712.779} C_VEL
LIN {X 0,Y 580.11,Z 721.531,A -85,B 0,C 180,E1 -1713.821,E2 -1713.821} C_VEL
LIN {X 0,Y 580.053,Z 717.63,A -85,B 0,C 180,E1 -1714.866,E2 -1714.866} C_VEL
LIN {X 0,Y 580.162,Z 712.597,A -85,B 0,C 180,E1 -1715.911,E2 -1715.911} C_VEL
LIN {X 0,Y 580.159,Z 706.274,A -85,B 0,C 180,E1 -1716.959,E2 -1716.959} C_VEL
LIN {X 0,Y 580.242,Z 698.353,A -85,B 0,C 180,E1 -1718.008,E2 -1718.008} C_VEL
LIN {X 0,Y 580.308,Z 688.503,A -85,B 0,C 180,E1 -1719.059,E2 -1719.059} C_VEL
LIN {X 0,Y 580.418,Z 678.179,A -85,B 0,C 180,E1 -1719.937,E2 -1719.937} C_VEL
LIN {X 0,Y 580.548,Z 666.544,A -85,B 0,C 180,E1 -1720.728,E2 -1720.728} C_VEL
LIN {X 0,Y 580.614,Z 654.977,A -85,B 0,C 180,E1 -1721.344,E2 -1721.344} C_VEL
LIN {X 0,Y 580.679,Z 642.972,A -85,B 0,C 180,E1 -1721.83,E2 -1721.83} C_VEL
LIN {X 0,Y 580.774,Z 629.932,A -85,B 0,C 180,E1 -1722.205,E2 -1722.205} C_VEL
LIN {X 0,Y 580.814,Z 617.571,A -85,B 0,C 180,E1 -1722.426,E2 -1722.426} C_VEL
LIN {X 0,Y 580.81,Z 518.194,A -85,B 0,C 180,E1 -1723.661,E2 -1723.661} C_VEL
LIN {X 0,Y 580.399,Z 515.221,A -85,B 0,C 180,E1 -1723.726,E2 -1723.726} C_VEL
LIN {X 0,Y 580.547,Z 494.062,A -85,B 0,C 180,E1 -1726.71,E2 -1726.71} C_VEL
LIN {X 0,Y 580.748,Z 473.561,A -85,B 0,C 180,E1 -1729.643,E2 -1729.643} C_VEL
LIN {X 0,Y 580.933,Z 454.604,A -85,B 0,C 180,E1 -1732.401,E2 -1732.401} C_VEL
LIN {X 0,Y 580.298,Z 449.828,A -85,B 0,C 180,E1 -1733.166,E2 -1733.166} C_VEL
LIN {X 0,Y 580.3,Z 449.829,A -85,B 0,C 180,E1 -1735.849,E2 -1735.849} C_VEL
LIN {X 0,Y 580.306,Z 449.823,A -85,B 0,C 180,E1 -1738.186,E2 -1738.186} C_VEL
LIN {X 0,Y 580.294,Z 449.822,A -85,B 0,C 180,E1 -1740.696,E2 -1740.696} C_VEL
LIN {X 0,Y 580.31,Z 449.823,A -85,B 0,C 180,E1 -1743.317,E2 -1743.317} C_VEL
LIN {X 0,Y 580.252,Z 449.835,A -85,B 0,C 180,E1 -1745.757,E2 -1745.757} C_VEL
LIN {X 0,Y 580.295,Z 449.823,A -85,B 0,C 180,E1 -1748.147,E2 -1748.147} C_VEL
LIN {X 0,Y 580.305,Z 449.819,A -85,B 0,C 180,E1 -1750.844,E2 -1750.844} C_VEL
LIN {X 0,Y 580.294,Z 449.83,A -85,B 0,C 180,E1 -1753.657,E2 -1753.657} C_VEL
LIN {X 0,Y 580.282,Z 449.822,A -85,B 0,C 180,E1 -1756.61,E2 -1756.61} C_VEL
LIN {X 0,Y 580.303,Z 449.821,A -85,B 0,C 180,E1 -1759.157,E2 -1759.157} C_VEL
LIN {X 0,Y 580.295,Z 449.826,A -85,B 0,C 180,E1 -1761.927,E2 -1761.927} C_VEL
LIN {X 0,Y 580.312,Z 449.819,A -85,B 0,C 180,E1 -1764.457,E2 -1764.457} C_VEL
LIN {X 0,Y 580.297,Z 449.821,A -85,B 0,C 180,E1 -1766.975,E2 -1766.975} C_VEL
LIN {X 0,Y 580.3,Z 449.825,A -85,B 0,C 180,E1 -1769.425,E2 -1769.425} C_VEL
LIN {X 0,Y 580.298,Z 449.823,A -85,B 0,C 180,E1 -1772.142,E2 -1772.142} C_VEL
LIN {X 0,Y 580.313,Z 449.82,A -85,B 0,C 180,E1 -1774.92,E2 -1774.92} C_VEL
LIN {X 0,Y 580.337,Z 449.863,A -85,B 0,C 180,E1 -1776.136,E2 -1776.136} C_VEL
LIN {X 0,Y 581.048,Z 455.337,A -85,B 0,C 180,E1 -1776.939,E2 -1776.939} C_VEL
LIN {X 0,Y 580.821,Z 476.167,A -85,B 0,C 180,E1 -1779.827,E2 -1779.827} C_VEL
LIN {X 0,Y 580.621,Z 496.407,A -85,B 0,C 180,E1 -1782.586,E2 -1782.586} C_VEL
LIN {X 0,Y 580.459,Z 518.176,A -85,B 0,C 180,E1 -1785.51,E2 -1785.51} C_VEL
LIN {X 0,Y 580.408,Z 524.674,A -85,B 0,C 180,E1 -1786.376,E2 -1786.376} C_VEL
LIN {X 0,Y 580.973,Z 528.882,A -85,B 0,C 180,E1 -1786.445,E2 -1786.445} C_VEL
LIN {X 0,Y 580.808,Z 632.925,A -85,B 0,C 180,E1 -1787.752,E2 -1787.752} C_VEL
LIN {X 0,Y 580.735,Z 645.675,A -85,B 0,C 180,E1 -1788.039,E2 -1788.039} C_VEL
LIN {X 0,Y 580.632,Z 659.441,A -85,B 0,C 180,E1 -1788.515,E2 -1788.515} C_VEL
LIN {X 0,Y 580.539,Z 671.563,A -85,B 0,C 180,E1 -1789.096,E2 -1789.096} C_VEL
LIN {X 0,Y 580.441,Z 681.725,A -85,B 0,C 180,E1 -1789.712,E2 -1789.712} C_VEL
LIN {X 0,Y 580.347,Z 692.262,A -85,B 0,C 180,E1 -1790.503,E2 -1790.503} C_VEL
LIN {X 0,Y 580.301,Z 702.575,A -85,B 0,C 180,E1 -1791.468,E2 -1791.468} C_VEL
LIN {X 0,Y 580.2,Z 711.535,A -85,B 0,C 180,E1 -1792.518,E2 -1792.518} C_VEL
LIN {X 0,Y 580.135,Z 717.749,A -85,B 0,C 180,E1 -1793.407,E2 -1793.407} C_VEL
LIN {X 0,Y 580.139,Z 723.632,A -85,B 0,C 180,E1 -1794.438,E2 -1794.438} C_VEL
LIN {X 0,Y 580.108,Z 728.375,A -85,B 0,C 180,E1 -1795.483,E2 -1795.483} C_VEL
LIN {X 0,Y 580.124,Z 732.017,A -85,B 0,C 180,E1 -1796.527,E2 -1796.527} C_VEL
LIN {X 0,Y 580.043,Z 733.893,A -85,B 0,C 180,E1 -1797.222,E2 -1797.222} C_VEL
LIN {X 0,Y 580.038,Z 735.344,A -85,B 0,C 180,E1 -1797.917,E2 -1797.917} C_VEL
LIN {X 0,Y 580.041,Z 736.965,A -85,B 0,C 180,E1 -1799.306,E2 -1799.306} C_VEL
LIN {X 0,Y 580.038,Z 737.206,A -85,B 0,C 180,E1 -1800,E2 -1800} C_VEL
LIN {X 0,Y 580.047,Z 736.442,A -85,B 0,C 180,E1 -1801.388,E2 -1801.388} C_VEL
LIN {X 0,Y 580.037,Z 735.488,A -85,B 0,C 180,E1 -1802.083,E2 -1802.083} C_VEL
LIN {X 0,Y 580.123,Z 732.289,A -85,B 0,C 180,E1 -1803.473,E2 -1803.473} C_VEL
LIN {X 0,Y 580.108,Z 728.741,A -85,B 0,C 180,E1 -1804.516,E2 -1804.516} C_VEL
LIN {X 0,Y 580.137,Z 724.096,A -85,B 0,C 180,E1 -1805.561,E2 -1805.561} C_VEL
LIN {X 0,Y 580.169,Z 718.132,A -85,B 0,C 180,E1 -1806.621,E2 -1806.621} C_VEL
LIN {X 0,Y 580.221,Z 710.887,A -85,B 0,C 180,E1 -1807.657,E2 -1807.657} C_VEL
LIN {X 0,Y 580.255,Z 701.775,A -85,B 0,C 180,E1 -1808.708,E2 -1808.708} C_VEL
LIN {X 0,Y 580.369,Z 691.225,A -85,B 0,C 180,E1 -1809.673,E2 -1809.673} C_VEL
LIN {X 0,Y 580.446,Z 681.753,A -85,B 0,C 180,E1 -1810.376,E2 -1810.376} C_VEL
LIN {X 0,Y 580.555,Z 671.596,A -85,B 0,C 180,E1 -1810.991,E2 -1810.991} C_VEL
LIN {X 0,Y 580.652,Z 659.695,A -85,B 0,C 180,E1 -1811.564,E2 -1811.564} C_VEL
LIN {X 0,Y 580.739,Z 645.729,A -85,B 0,C 180,E1 -1812.049,E2 -1812.049} C_VEL
LIN {X 0,Y 580.78,Z 633.013,A -85,B 0,C 180,E1 -1812.337,E2 -1812.337} C_VEL
LIN {X 0,Y 580.829,Z 527.627,A -85,B 0,C 180,E1 -1813.664,E2 -1813.664} C_VEL
LIN {X 0,Y 580.423,Z 524.598,A -85,B 0,C 180,E1 -1813.724,E2 -1813.724} C_VEL
LIN {X 0,Y 580.581,Z 503.644,A -85,B 0,C 180,E1 -1816.527,E2 -1816.527} C_VEL
LIN {X 0,Y 580.783,Z 480.691,A -85,B 0,C 180,E1 -1819.642,E2 -1819.642} C_VEL
LIN {X 0,Y 580.999,Z 459.387,A -85,B 0,C 180,E1 -1822.585,E2 -1822.585} C_VEL
LIN {X 0,Y 580.889,Z 452.681,A -85,B 0,C 180,E1 -1823.532,E2 -1823.532} C_VEL
LIN {X 0,Y 580.312,Z 449.827,A -85,B 0,C 180,E1 -1823.983,E2 -1823.983} C_VEL
LIN {X 0,Y 580.282,Z 449.828,A -85,B 0,C 180,E1 -1826.623,E2 -1826.623} C_VEL
LIN {X 0,Y 580.307,Z 449.82,A -85,B 0,C 180,E1 -1829.31,E2 -1829.31} C_VEL
LIN {X 0,Y 580.303,Z 449.829,A -85,B 0,C 180,E1 -1832.2,E2 -1832.2} C_VEL
LIN {X 0,Y 580.305,Z 449.821,A -85,B 0,C 180,E1 -1834.695,E2 -1834.695} C_VEL
LIN {X 0,Y 580.304,Z 449.82,A -85,B 0,C 180,E1 -1837.268,E2 -1837.268} C_VEL
LIN {X 0,Y 580.296,Z 449.825,A -85,B 0,C 180,E1 -1840.27,E2 -1840.27} C_VEL
LIN {X 0,Y 580.28,Z 449.823,A -85,B 0,C 180,E1 -1842.706,E2 -1842.706} C_VEL
LIN {X 0,Y 580.276,Z 449.83,A -85,B 0,C 180,E1 -1845.609,E2 -1845.609} C_VEL
LIN {X 0,Y 580.294,Z 449.823,A -85,B 0,C 180,E1 -1848.232,E2 -1848.232} C_VEL
LIN {X 0,Y 580.282,Z 449.823,A -85,B 0,C 180,E1 -1850.965,E2 -1850.965} C_VEL
LIN {X 0,Y 580.273,Z 449.833,A -85,B 0,C 180,E1 -1853.596,E2 -1853.596} C_VEL
LIN {X 0,Y 580.32,Z 449.82,A -85,B 0,C 180,E1 -1856.145,E2 -1856.145} C_VEL
LIN {X 0,Y 580.281,Z 449.823,A -85,B 0,C 180,E1 -1858.614,E2 -1858.614} C_VEL
LIN {X 0,Y 580.297,Z 449.825,A -85,B 0,C 180,E1 -1861.023,E2 -1861.023} C_VEL
LIN {X 0,Y 580.295,Z 449.828,A -85,B 0,C 180,E1 -1863.666,E2 -1863.666} C_VEL
LIN {X 0,Y 580.345,Z 449.968,A -85,B 0,C 180,E1 -1865.39,E2 -1865.39} C_VEL
LIN {X 0,Y 581.387,Z 454.288,A -85,B 0,C 180,E1 -1865.921,E2 -1865.921} C_VEL
LIN {X 0,Y 581.219,Z 474.62,A -85,B 0,C 180,E1 -1868.171,E2 -1868.171} C_VEL
LIN {X 0,Y 580.938,Z 500.031,A -85,B 0,C 180,E1 -1870.934,E2 -1870.934} C_VEL
LIN {X 0,Y 580.723,Z 523.326,A -85,B 0,C 180,E1 -1873.431,E2 -1873.431} C_VEL
LIN {X 0,Y 581.413,Z 528.553,A -85,B 0,C 180,E1 -1873.519,E2 -1873.519} C_VEL
LIN {X 0,Y 581.121,Z 662.845,A -85,B 0,C 180,E1 -1875.219,E2 -1875.219} C_VEL
LIN {X 0,Y 581.037,Z 677.552,A -85,B 0,C 180,E1 -1875.559,E2 -1875.559} C_VEL
LIN {X 0,Y 580.926,Z 691.818,A -85,B 0,C 180,E1 -1876.042,E2 -1876.042} C_VEL
LIN {X 0,Y 580.812,Z 704.624,A -85,B 0,C 180,E1 -1876.619,E2 -1876.619} C_VEL
LIN {X 0,Y 580.657,Z 717.085,A -85,B 0,C 180,E1 -1877.327,E2 -1877.327} C_VEL
LIN {X 0,Y 580.527,Z 729.629,A -85,B 0,C 180,E1 -1878.211,E2 -1878.211} C_VEL
LIN {X 0,Y 580.442,Z 740.9,A -85,B 0,C 180,E1 -1879.189,E2 -1879.189} C_VEL
LIN {X 0,Y 580.276,Z 750.844,A -85,B 0,C 180,E1 -1880.237,E2 -1880.237} C_VEL
LIN {X 0,Y 580.241,Z 759.165,A -85,B 0,C 180,E1 -1881.291,E2 -1881.291} C_VEL
LIN {X 0,Y 580.166,Z 767.121,A -85,B 0,C 180,E1 -1882.517,E2 -1882.517} C_VEL
LIN {X 0,Y 580.093,Z 773.523,A -85,B 0,C 180,E1 -1883.739,E2 -1883.739} C_VEL
LIN {X 0,Y 580.078,Z 777.958,A -85,B 0,C 180,E1 -1884.786,E2 -1884.786} C_VEL
LIN {X 0,Y 580.102,Z 781.44,A -85,B 0,C 180,E1 -1885.831,E2 -1885.831} C_VEL
LIN {X 0,Y 580.041,Z 784.83,A -85,B 0,C 180,E1 -1887.221,E2 -1887.221} C_VEL
LIN {X 0,Y 580.041,Z 786.831,A -85,B 0,C 180,E1 -1888.611,E2 -1888.611} C_VEL
LIN {X 0,Y 580.036,Z 787.5,A -85,B 0,C 180,E1 -1889.999,E2 -1889.999} C_VEL
LIN {X 0,Y 580.041,Z 786.833,A -85,B 0,C 180,E1 -1891.388,E2 -1891.388} C_VEL
LIN {X 0,Y 580.041,Z 784.835,A -85,B 0,C 180,E1 -1892.777,E2 -1892.777} C_VEL
LIN {X 0,Y 580.102,Z 781.446,A -85,B 0,C 180,E1 -1894.168,E2 -1894.168} C_VEL
LIN {X 0,Y 580.128,Z 776.572,A -85,B 0,C 180,E1 -1895.561,E2 -1895.561} C_VEL
LIN {X 0,Y 580.14,Z 770.057,A -85,B 0,C 180,E1 -1896.957,E2 -1896.957} C_VEL
LIN {X 0,Y 580.192,Z 762.806,A -85,B 0,C 180,E1 -1898.182,E2 -1898.182} C_VEL
LIN {X 0,Y 580.286,Z 753.831,A -85,B 0,C 180,E1 -1899.409,E2 -1899.409} C_VEL
LIN {X 0,Y 580.356,Z 744.402,A -85,B 0,C 180,E1 -1900.465,E2 -1900.465} C_VEL
LIN {X 0,Y 580.474,Z 734.33,A -85,B 0,C 180,E1 -1901.403,E2 -1901.403} C_VEL
LIN {X 0,Y 580.618,Z 722.446,A -85,B 0,C 180,E1 -1902.317,E2 -1902.317} C_VEL
LIN {X 0,Y 580.729,Z 709.666,A -85,B 0,C 180,E1 -1903.114,E2 -1903.114} C_VEL
LIN {X 0,Y 580.91,Z 697.182,A -85,B 0,C 180,E1 -1903.734,E2 -1903.734} C_VEL
LIN {X 0,Y 581.017,Z 684.28,A -85,B 0,C 180,E1 -1904.233,E2 -1904.233} C_VEL
LIN {X 0,Y 581.079,Z 670.239,A -85,B 0,C 180,E1 -1904.629,E2 -1904.629} C_VEL
LIN {X 0,Y 581.156,Z 655.68,A -85,B 0,C 180,E1 -1904.89,E2 -1904.89} C_VEL
LIN {X 0,Y 581.323,Z 526.913,A -85,B 0,C 180,E1 -1906.504,E2 -1906.504} C_VEL
LIN {X 0,Y 580.73,Z 523.199,A -85,B 0,C 180,E1 -1906.582,E2 -1906.582} C_VEL
LIN {X 0,Y 581.012,Z 494.648,A -85,B 0,C 180,E1 -1909.647,E2 -1909.647} C_VEL
LIN {X 0,Y 581.271,Z 469.553,A -85,B 0,C 180,E1 -1912.386,E2 -1912.386} C_VEL
LIN {X 0,Y 581.383,Z 454.306,A -85,B 0,C 180,E1 -1914.077,E2 -1914.077} C_VEL
LIN {X 0,Y 580.333,Z 449.825,A -85,B 0,C 180,E1 -1914.652,E2 -1914.652} C_VEL
LIN {X 0,Y 580.318,Z 449.818,A -85,B 0,C 180,E1 -1917.862,E2 -1917.862} C_VEL
LIN {X 0,Y 580.298,Z 449.829,A -85,B 0,C 180,E1 -1920.696,E2 -1920.696} C_VEL
LIN {X 0,Y 580.301,Z 449.821,A -85,B 0,C 180,E1 -1923.316,E2 -1923.316} C_VEL
LIN {X 0,Y 580.322,Z 449.815,A -85,B 0,C 180,E1 -1925.767,E2 -1925.767} C_VEL
LIN {X 0,Y 580.285,Z 449.824,A -85,B 0,C 180,E1 -1928.145,E2 -1928.145} C_VEL
LIN {X 0,Y 580.315,Z 449.826,A -85,B 0,C 180,E1 -1930.84,E2 -1930.84} C_VEL
LIN {X 0,Y 580.284,Z 449.821,A -85,B 0,C 180,E1 -1933.656,E2 -1933.656} C_VEL
LIN {X 0,Y 580.278,Z 449.831,A -85,B 0,C 180,E1 -1936.607,E2 -1936.607} C_VEL
LIN {X 0,Y 580.296,Z 449.822,A -85,B 0,C 180,E1 -1939.156,E2 -1939.156} C_VEL
LIN {X 0,Y 580.283,Z 449.822,A -85,B 0,C 180,E1 -1941.926,E2 -1941.926} C_VEL
LIN {X 0,Y 580.302,Z 449.824,A -85,B 0,C 180,E1 -1944.456,E2 -1944.456} C_VEL
LIN {X 0,Y 580.285,Z 449.826,A -85,B 0,C 180,E1 -1946.975,E2 -1946.975} C_VEL
LIN {X 0,Y 580.301,Z 449.819,A -85,B 0,C 180,E1 -1949.425,E2 -1949.425} C_VEL
LIN {X 0,Y 580.311,Z 449.82,A -85,B 0,C 180,E1 -1952.136,E2 -1952.136} C_VEL
LIN {X 0,Y 580.301,Z 449.824,A -85,B 0,C 180,E1 -1954.92,E2 -1954.92} C_VEL
LIN {X 0,Y 580.268,Z 449.821,A -85,B 0,C 180,E1 -1957.947,E2 -1957.947} C_VEL
LIN {X 0,Y 580.307,Z 449.824,A -85,B 0,C 180,E1 -1960.914,E2 -1960.914} C_VEL
LIN {X 0,Y 580.275,Z 449.822,A -85,B 0,C 180,E1 -1963.826,E2 -1963.826} C_VEL
LIN {X 0,Y 580.274,Z 449.831,A -85,B 0,C 180,E1 -1966.696,E2 -1966.696} C_VEL
LIN {X 0,Y 580.297,Z 449.819,A -85,B 0,C 180,E1 -1969.533,E2 -1969.533} C_VEL
LIN {X 0,Y 580.331,Z 449.822,A -85,B 0,C 180,E1 -1972.345,E2 -1972.345} C_VEL
LIN {X 0,Y 580.337,Z 449.817,A -85,B 0,C 180,E1 -1975.137,E2 -1975.137} C_VEL
LIN {X 0,Y 580.329,Z 449.816,A -85,B 0,C 180,E1 -1977.918,E2 -1977.918} C_VEL
LIN {X 0,Y 580.36,Z 449.82,A -85,B 0,C 180,E1 -1980.694,E2 -1980.694} C_VEL
LIN {X 0,Y 580.281,Z 449.821,A -85,B 0,C 180,E1 -1983.472,E2 -1983.472} C_VEL
LIN {X 0,Y 580.315,Z 449.817,A -85,B 0,C 180,E1 -1985.56,E2 -1985.56} C_VEL
LIN {X 0,Y 580.327,Z 449.822,A -85,B 0,C 180,E1 -1988.356,E2 -1988.356} C_VEL
LIN {X 0,Y 580.322,Z 449.818,A -85,B 0,C 180,E1 -1991.209,E2 -1991.209} C_VEL
LIN {X 0,Y 580.304,Z 449.825,A -85,B 0,C 180,E1 -1994.339,E2 -1994.339} C_VEL
LIN {X 0,Y 580.304,Z 449.822,A -85,B 0,C 180,E1 -1996.915,E2 -1996.915} C_VEL
LIN {X 0,Y 580.3,Z 449.82,A -85,B 0,C 180,E1 -1999.823,E2 -1999.823} C_VEL
LIN {X 0,Y 580.278,Z 449.822,A -85,B 0,C 180,E1 -2001.345,E2 -2001.345} C_VEL
LIN {X 0,Y 579.581,Z 449.911,A -85,B 0,C 180,E1 -2001.925,E2 -2001.925} C_VEL
LIN {X 0,Y 576.703,Z 450.272,A -85,B 0,C 180,E1 -2002.864,E2 -2002.864} C_VEL
